# B&R Automation Studio project Soiled_PLC (part 6)

#### 12_sp2Cyclic.ab
```automation-basic
PROGRAM _CYCLIC
	(* cyclic program *)

;---------------------------------------
;Sequence 12 - SP2 Single point 2 D[912]
;---------------------------------------

;Inputs

I_BagAtBuffer			= X[9].X08
I_PaddleInPosition		= X[9].X10
I_BagInIncline			= X[9].X09
;I_BagOutAtTop           = X[7].X13

InclineEnable 		= ((D[17] > 0) AND NOT Std.HaltSys)

O_OpenBufferStop		= FALSE
O_RunMotor 				= FALSE

I_BagAtOutgoingBuffer	= FALSE
O_OutgoingBufferOpen	= FALSE

Alarm[17].Name 			= 0
Alarm[17].Bag			= 10005
Alarm[17].Beacon		= TRUE
Alarm[17].Extra			= 0
Alarm[17].Time			= 3000

;Setup Sequence
STEP = D[917]
;Setup Pulse contact
PLS = (STEP <> LASTSTEP)
LASTSTEP = STEP

;Sequence
;Step 0 - Disabled
IF (STEP = 0) THEN
	;Disabled
ENDIF

;Run Incline until paddle in position
IF (STEP = 1) THEN
	O_RunMotor = NOT I_PaddleInPosition
	IF I_PaddleInPosition THEN
		D[917] = 2
	ENDIF
	IF NOT Std.EStop THEN
		Alarm[17].Name = almSwitchFault
	ENDIF
ENDIF

;Wait for at buffer
TON_10ms(I_BagAtBuffer,300,BagAtBuffer,BagAtBufferET)
IF (STEP = 2) THEN
	IF (BagAtBuffer  AND NOT Std.HaltSys AND (D[17]>0)) THEN
		D[917] = 3
	ENDIF
	;IF (Bag[266].Cat > 0) AND NOT I_BagAtBuffer THEN
		;Alarm[12].Name 	= almBagNotAtProx
		;Alarm[12].Bag	= 266
	;ELSE IF (Bag[266].Cat = 0) AND I_BagAtBuffer THEN
		;Alarm[12].Name 	= almBagNotShownOnScreen
		;Alarm[12].Bag	= 266
	;ENDIF
ENDIF

;Open Buffer stop
IF (STEP = 3) THEN
	O_OpenBufferStop 	= TRUE
	;Enable.SIC[1]		= NOT I_BagInIncline
	IF I_BagInIncline THEN
		D[917] = 4
	ENDIF
	Alarm[17].Name = almBagNotArrived
ENDIF

;Let bag settle at base of incline
TON_10ms((STEP = 4),300,BagSettled,BagSettledET)
IF (STEP = 4) THEN
	;O_OpenBufferStop 	= TRUE
	;IF PLS THEN
	;	Bag[265] = Bag[266]
	;	Bag[266] = Bag[0]
	;ENDIF
	IF BagSettled THEN
		D[917] = 5
	ENDIF
ENDIF

;Move Bag up incline
TON_10ms((STEP = 5),700,BagNearTop,BagNearTopET)
TON_10ms(((STEP = 5) AND NOT I_BagInIncline),1000,CloseBufferStop,CloseBufferStopET)
IF (STEP = 5) THEN
	;O_OpenBufferStop 	= NOT CloseBufferStop
	O_RunMotor 			= NOT BagNearTop
	IF BagNearTop THEN
		D[917] = 6
	ENDIF
	Alarm[17].Name = almSwitchFault
ENDIF

;Check for space at destination
;Run motor for 0.5 seconds
TON_10ms((STEP = 6),50,RunOn,RunOnET)
IF (STEP = 6) THEN
	O_RunMotor 		= NOT RunOn

	IF Line[27].Clear THEN
		C[27] = 0
		D[917] = 7
	ENDIF
ENDIF

;Run incline until bag released / arrive at buffer
IF (STEP = 7) THEN
	O_RunMotor 			= TRUE
	;IF PLS THEN
	;	C[13] = 0
	;ENDIF
	IF Line[27].Trip THEN
		D[917] = 1
	ENDIF
	Alarm[17].Name = almBagNotReleased
ENDIF

;Alarms
TimerAlarm.IN 	= NOT PLS AND (Alarm[17].Name > 0)
TimerAlarm.PT 	= Alarm[17].Time
TimerAlarm FUB TON_10ms()
Alarm[17].On 	= TimerAlarm.Q
Alarm[17].ET 	= TimerAlarm.ET

;Outputs
Y[9].Y08 = O_OpenBufferStop
Y[13].Y14 = O_RunMotor
END_PROGRAM
```

### Program Logical/Sequences/10ms/18_sp6 (IEC) - * SP2 Empty bags from SDC1/2

#### 12_sp2.var
```iecst
VAR RETAIN
	STEP : UINT;
	PLS : BOOL;
	LASTSTEP : UINT;
END_VAR
VAR
	TimerAlarm : TON_10ms;
	I_BagAtBuffer : BOOL;
	O_OpenBuffer : BOOL;
	SDC2BufferFullET : TIME;
	SDC2BufferFull : BOOL;
	SettledBufferET : TIME;
	SettledBuffer : BOOL;
	O_OpenSP2BufferStop : BOOL;
	O_SelectPoint : BOOL;
	SP2BufferFull : BOOL;
	SP2BufferFullET : UDINT;
	ParingLoopEnabled : BOOL;
	BagInLoopHasDest : BOOL;
	BagAtBuffer : BOOL;
	SettledBufferSVC1 : BOOL;
	SettledBufferSVC1ET : UDINT;
	SettledBufferSVC2 : BOOL;
	SettledBufferSVC2ET : UDINT;
	O_SelectPointSVC1 : BOOL;
	O_SelectPointSVC2 : BOOL;
	I_BagatBuffer : BOOL;
	I_BagAtSVC1BufferStop : BOOL;
	I_BagAtSVC2BufferStop : BOOL;
	O_SVC1BufferStop : BOOL;
	O_SVC2BufferStop : BOOL;
	O_SelectSVC1 : BOOL;
	O_SelectSVC2 : BOOL;
	Alernate : USINT;
	BagAtBufferET : UDINT;
END_VAR
```

#### 12_sp2Cyclic.ab
```automation-basic
PROGRAM _CYCLIC
	(* cyclic program *)

;---------------------------------------
;Sequence 8 - SP8 Single point 2 D[912]
;---------------------------------------

;Inputs

I_BagatBuffer			= X[8].X11
I_BagAtSVC1BufferStop   = X[3].X06
I_BagAtSVC2BufferStop   = X[3].X14

O_SVC1BufferStop        = Y[3].Y06
O_SVC2BufferStop        = Y[3].Y14

O_OpenBuffer			= FALSE ;YB12
O_SelectSVC1            = FALSE ;YB11
O_SelectSVC2            = FALSE ;YB10

Alarm[18].Name 			= 0
Alarm[18].Bag			= 10006
Alarm[18].Beacon		= TRUE
Alarm[18].Extra			= 0
Alarm[18].Time			= 3000

;Setup Sequence
STEP = D[918]
;Setup Pulse contact
PLS = (STEP <> LASTSTEP)
LASTSTEP = STEP

;Sequence
;Step 0 - Disabled
IF (STEP = 0) THEN
	;Disabled
ENDIF

;Step 1 - decide where to take bag from
TON_10ms(I_BagatBuffer,300,BagAtBuffer,BagAtBufferET)
IF (STEP = 1) THEN

	IF BagAtBuffer THEN
	IF (Alernate > 2) THEN
		Alernate = 0
	ENDIF
	Alernate = Alernate + 1
			IF ((Alernate = 1)AND Line[28].Clear AND NOT I_BagAtSVC1BufferStop AND NOT O_SVC1BufferStop) THEN
				C[28]  = 0
				D[918] = 2
			ELSE IF ((Alernate = 2)AND Line[29].Clear AND NOT I_BagAtSVC2BufferStop AND NOT O_SVC2BufferStop) THEN
				C[29]  = 0
				D[918] = 3
			ENDIF
	ENDIF
ENDIF

;Step 2 - Bag from svc1
IF (STEP = 2) THEN
	O_OpenBuffer = TRUE
	O_SelectSVC1 = TRUE
	IF Line[28].Trip THEN
		D[918] = 1
	ENDIF
	Alarm[18].Name = almBagNotArrived
ENDIF

;Step 2 - Bag from svc1
IF (STEP = 3) THEN
	O_OpenBuffer = TRUE
	O_SelectSVC2 = TRUE
	IF Line[29].Trip THEN
		D[918] = 1
	ENDIF
	Alarm[8].Name = almBagNotArrived
ENDIF

;Alarms
TimerAlarm.IN 	= NOT PLS AND (Alarm[18].Name > 0)
TimerAlarm.PT 	= Alarm[18].Time
TimerAlarm FUB TON_10ms()
Alarm[18].On 	= TimerAlarm.Q
Alarm[18].ET 	= TimerAlarm.ET

;Outputs
Y[8].Y11 = O_OpenBuffer
Y[8].Y12 = O_SelectSVC1
Y[8].Y13 = O_SelectSVC2
END_PROGRAM
```

### Program Logical/Sequences/10ms/19_sp7 (IEC) - * SP2 Empty bags from SDC1/2

#### 12_sp2.var
```iecst
VAR RETAIN
	STEP : UINT;
	PLS : BOOL;
	LASTSTEP : UINT;
END_VAR
VAR
	TimerAlarm : TON_10ms;
	I_BagAtBuffer : BOOL;
	O_OpenBuffer : BOOL;
	SDC2BufferFullET : TIME;
	SDC2BufferFull : BOOL;
	SettledBufferET : TIME;
	SettledBuffer : ARRAY[0..2] OF BOOL;
	O_OpenSP2BufferStop : BOOL;
	O_SelectPoint : BOOL;
	SP2BufferFull : BOOL;
	SP2BufferFullET : UDINT;
	ParingLoopEnabled : BOOL;
	BagInLoopHasDest : BOOL;
	O_OpenSDC1BufferStop : BOOL;
	BagSettledAtBuffer : BOOL;
	BagSettledAtBufferET : UDINT;
	Alternator : USINT;
	BagAtBuffer : ARRAY[0..2] OF BOOL;
	SettledBufferDC1 : BOOL;
	SettledBufferDC1ET : UDINT;
	SettledBufferSD2 : BOOL;
	SettledBufferDC2ET : UDINT;
	SettledBufferDC2 : BOOL;
	I_BagAtSVC1BufferStop : BOOL;
	I_BagAtSVC2BufferStop : BOOL;
	Reset : BOOL;
	ResetET : UDINT;
	BagAtSVC1BufferStop : BOOL;
	BagAtSVC1BufferStopET : UDINT;
	BagAtSVC2BufferStop : BOOL;
	BagAtSVC2BufferStopET : UDINT;
	Alernate : USINT;
	O_SelectSVC1 : BOOL;
	O_SelectSVC2 : BOOL;
END_VAR
```

#### 12_sp2Cyclic.ab
```automation-basic
PROGRAM _CYCLIC
	(* cyclic program *)

;---------------------------------------
;Sequence 12 - SP2 Single point 2 D[912]
;---------------------------------------

;Inputs

I_BagAtSVC1BufferStop   = X[9].X05
I_BagAtSVC2BufferStop   = X[9].X06

O_OpenSDC1BufferStop	= FALSE
O_SelectPoint       	           = FALSE
O_SelectSVC1                      = FALSE
O_SelectSVC2                      = FALSE

Alarm[19].Name 			= 0
Alarm[19].Bag			= 10012
Alarm[19].Beacon	    = TRUE
Alarm[19].Extra			= 0
Alarm[19].Time			= 3000

;Setup Sequence
STEP = D[919]
;Setup Pulse contact

PLS = (STEP <> LASTSTEP)
LASTSTEP = STEP

;Sequence
;Step 0 - Disabled
IF (STEP = 0) THEN
	;Disabled
ENDIF

;Step 1 - decide where to take bag from
TON_10ms((STEP = 1),300,Reset,ResetET)
IF (STEP = 1) THEN

	IF Reset THEN
		D[919] = 2
	ENDIF
ENDIF

;Wait for Bag at buffer and destination clear
TON_10ms(I_BagAtSVC1BufferStop,300,BagAtSVC1BufferStop,BagAtSVC1BufferStopET)
TON_10ms(I_BagAtSVC2BufferStop,300,BagAtSVC2BufferStop,BagAtSVC2BufferStopET)
IF (STEP = 2) THEN
	IF (Request.SP[7] = TRUE) THEN
	IF (Alernate > 2) THEN
		Alernate = 0
	ENDIF
	Alernate = Alernate + 1
			IF ((Alernate = 1)AND BagAtSVC1BufferStop) THEN
				D[919] = 3
			ELSE IF ((Alernate = 2)AND BagAtSVC2BufferStop) THEN
				D[919] = 4
			ENDIF
	ENDIF
ENDIF

;Enable release
IF ((STEP = 3) OR (STEP = 4)) THEN
		Enable.SP[7] = TRUE
	ELSE
		Enable.SP[7] = FALSE
ENDIF

;Open buffer stop and point
IF (STEP = 3) THEN
	O_SelectSVC1 = TRUE
	IF (NOT Request.SP[7]) THEN
		D[919] = 1
	ENDIF
	Alarm[19].Name = almBagNotArrived
ENDIF

;select svc 2 point and stop
IF (STEP = 4) THEN
	O_SelectSVC2 = TRUE
	IF (NOT Request.SP[7]) THEN
		D[919] = 1
	ENDIF
	Alarm[9].Name = almBagNotArrived
ENDIF
;Alarms
TimerAlarm.IN 	= NOT PLS AND (Alarm[19].Name > 0)
TimerAlarm.PT 	= Alarm[19].Time
TimerAlarm FUB TON_10ms()
Alarm[19].On 	= TimerAlarm.Q
Alarm[19].ET 	= TimerAlarm.ET

;Outputs
Y[9].Y05 = O_SelectSVC1
Y[9].Y06 = O_SelectSVC2
END_PROGRAM
```

### Program Logical/Sequences/10ms/20_sp1 (IEC) - * SP2 Empty bags from SDC1/2

#### 12_sp2.var
```iecst
VAR RETAIN
	STEP : UINT;
	PLS : BOOL;
	LASTSTEP : UINT;
END_VAR
VAR
	TimerAlarm : TON_10ms;
	I_BagAtBuffer : BOOL;
	O_OpenBuffer : BOOL;
	SDC2BufferFullET : TIME;
	SDC2BufferFull : BOOL;
	SettledBufferET : TIME;
	SettledBuffer : BOOL;
	O_OpenSP2BufferStop : BOOL;
	O_SelectPoint : BOOL;
	SP2BufferFull : BOOL;
	SP2BufferFullET : UDINT;
	ParingLoopEnabled : BOOL;
	BagInLoopHasDest : BOOL;
	BagAtBuffer : BOOL;
	SettledBufferSVC1 : BOOL;
	SettledBufferSVC1ET : UDINT;
	SettledBufferSVC2 : BOOL;
	SettledBufferSVC2ET : UDINT;
	O_SelectPointSVC1 : BOOL;
	O_SelectPointSVC2 : BOOL;
	Reset : BOOL;
	ResetET : UDINT;
	I_BagatBuffer : BOOL;
	BagAtBufferET : UDINT;
	Alernate : USINT;
	I_BagAtSVC1BufferStop : BOOL;
	O_SVC1BufferStop : BOOL;
	I_BagAtSVC2BufferStop : BOOL;
	O_SVC2BufferStop : BOOL;
	O_SelectSVC1 : BOOL;
	O_SelectSVC2 : BOOL;
END_VAR
```

#### 12_sp2Cyclic.ab
```automation-basic
PROGRAM _CYCLIC
	(* cyclic program *)

;---------------------------------------
;Sequence 8 - SP8 Single point 2 D[912]
;---------------------------------------

;Inputs

O_SelectSVC1              = FALSE ;YB11
O_SelectSVC2              = FALSE ;YB10

Alarm[20].Name 			= 0
Alarm[20].Bag			= 221
Alarm[20].Beacon		= TRUE
Alarm[20].Extra			= 0
Alarm[20].Time			= 5000

;Setup Sequence
STEP = D[920]
;Setup Pulse contact
PLS = (STEP <> LASTSTEP)
LASTSTEP = STEP

;Sequence
;Step 0 - Disabled
IF (STEP = 0) THEN
	;Disabled
ENDIF

;clear data
TON_10ms((STEP = 1),100,Reset,ResetET)
IF (STEP = 1) THEN
	IF (Reset = TRUE)and (Bag[221].Cat = 0) THEN
		D[920] = 2
	ENDIF
ENDIF

;Wait SLU1 request and destination clear
TON_10ms(I_BagatBuffer,300,BagAtBuffer,BagAtBufferET)
IF (STEP = 2) THEN
	IF (Request.LU[1] = TRUE) THEN
	IF (Alernate > 2) THEN
		Alernate = 0
	ENDIF
	Alernate = Alernate + 1
			IF ((Alernate = 1)AND Line[30].Clear AND (Bag[223].Cat =0) AND NOT I_BagAtSVC1BufferStop AND NOT O_SVC1BufferStop) THEN
				C[30]  = 0
				D[45]  = 1
				D[920] = 3
			ELSE IF ((Alernate = 2)AND Line[18].Clear AND (Bag[222].Cat =0) AND NOT I_BagAtSVC2BufferStop AND NOT O_SVC2BufferStop) THEN
				C[18]  = 0
				D[45]  = 2
				D[920] = 4
			ENDIF
	ENDIF
ENDIF

;enable slu1 to release
IF ((STEP = 3) OR (STEP = 4)) THEN
	Enable.LU[1] = TRUE
	ELSE
	Enable.LU[1] = FALSE
ENDIF

;Open buffer to release a bag to svc 1
IF (STEP = 3) THEN

	O_SelectSVC1 = TRUE

	IF Line[30].Trip THEN
		IF (Bag[221].Cat > 0) AND (Bag[223].Cat= 0) THEN
			Bag[223] = Bag[221]
			Bag[221] = Bag[0]
		ENDIF
			D[920] = 1
	ENDIF
	Alarm[20].Name 	= almBagNotArrived
ENDIF

;select svc 2 point
IF (STEP = 4) THEN
O_SelectSVC2 = TRUE

	IF Line[18].Trip THEN
		IF (Bag[221].Cat > 0) AND (Bag[222].Cat= 0) THEN
			Bag[222] = Bag[221]
			Bag[221] = Bag[0]
		ENDIF
		D[920] = 1
	ENDIF
	Alarm[20].Name 	= almBagNotArrived
ENDIF

;Outputs

Y[9].Y07 = O_SelectSVC1
Y[9].Y12 = O_SelectSVC2

;Alarms
TimerAlarm.IN 	= NOT PLS AND (Alarm[20].Name > 0)
TimerAlarm.PT 	= Alarm[20].Time
TimerAlarm FUB TON_10ms()
Alarm[20].On 	= TimerAlarm.Q
Alarm[20].ET 	= TimerAlarm.ET

;Outputs
;Y[6].Y07 = O_SelectPointSVC1
;Y[6].Y08 = O_SelectPointSVC2
END_PROGRAM
```

### Program Logical/Sequences/10ms/10_sb1_ref (IEC, version 2.00.0) - *FROM OLD PROGRAM__ REF ONLY

#### 2_belt1Cyclic.ab
```automation-basic
PROGRAM _CYCLIC
 	(* cyclic program *)

;Sequence 2 - Transfer Belt 1 from Stations 1-12

;-----------------------------------------
;Revision 1.00 18/01/2006 D.J. First Issue
;-----------------------------------------

;Inputs and Outputs
;------------------

;Bank 						= 1

I_PhotoBottomSDC1LoadDropped = X[3].X09
I_PhotoMiddleBelt  			 = X[3].X12
I_PhotocellAtEnd             = X[5].X16
I_OpenBag                    = X[3].X05
I_LoadDropped                = X[3].X06

Enable.SDC1Drop          	= FALSE

O_RunBelt 					= FALSE
O_BagReady                  = FALSE

Alarm[10].Name 				= 0
Alarm[10].Bag				= 160
Alarm[10].Beacon			= TRUE
Alarm[10].Extra				= 0
Alarm[10].Time				= 5000

STEP = D[910]
;Setup Pulse contact
PLS = (STEP <> LASTSTEP)
LASTSTEP = STEP

;Step 0 - Disabled
IF STEP = 0 THEN
	;Disabled
ENDIF

;Step 1 - Run belt till clear
TON_10ms(((STEP = 1) AND NOT I_PhotoBottomSDC1LoadDropped AND NOT I_PhotoMiddleBelt AND NOT I_PhotocellAtEnd),500,BeltClear,BeltClearET)
IF STEP = 1 THEN
	O_RunBelt = TRUE
	IF BeltClear THEN

			D[910] = 2 ;No Bag on belt

	ENDIF
	Alarm[10].Time = 10000
	Alarm[10].Name = almPhotocellBlocked
ENDIF

;Step 2 - Wait for SDC 1 to request to drop
IF STEP = 2 THEN

		;------Write Report------
		IF Std.StationReports  THEN

			IF (ReportLoading[n].Cat = 0) THEN

				;Check if anything has been added and current weight is not less than the previous
				WeightValue = Stn[n].Weight - INT(StnPrev[n].Wgt)
				WeightValid = (WeightValue > 0)

				IF WeightValid THEN

					;Ensure valid values as we report on either a weight or count change
					IF (WeightValue < 0) THEN
						WeightValue = 0
					ENDIF

					ReportLoading[n].Cat = UINT(Bag[StnBag].Cat)	;Category
					ReportLoading[n].Cus = Bag[StnBag].Cus			;Customer
					ReportLoading[n].Wgt = UINT(WeightValue)		;Weight
					ReportLoading[n].Cnt = 0						;Count
					ReportLoading[n].Stn = n         				;Station
					ReportLoading[n].Mcn = 0						;Machine

				ENDIF

			ENDIF

		ENDIF
		IF Request.SDC1Drop THEN
			D[910] = 3
		ENDIF

		Alarm[10].Name = almNoAlarm

ENDIF

;Step 3
;Open Bag and Release to Belt Conveyor
IF STEP = 3 THEN
	Enable.SDC1Drop = TRUE
	O_RunBelt       = TRUE
	IF I_PhotoBottomSDC1LoadDropped THEN
		Bag[160] = Bag[151]

	ENDIF
	IF (Bag[160].Cat > 0) AND NOT Request.SDC1Drop AND I_PhotoBottomSDC1LoadDropped THEN
		D[910] = 4
	ENDIF
	Alarm[10].Name = almLoadNotDropped
ENDIF

;Step 4 - Run Belt Till middle
IF STEP = 4 THEN
	O_RunBelt = TRUE
	IF I_PhotoMiddleBelt THEN
		D[910] = 5
	ENDIF
	;Alarm[2].Name = almNoAlarm
ENDIF

;Step 5 - Check second bag is pair
IF STEP = 5 THEN
	;O_RunBelt = TRUE
	IF Request.SDC1Drop AND (Bag[151].Cat = Bag[160].Cat) THEN
		Bag[160].Wgt = Bag[160].Wgt + Bag[151].Wgt
		D[910] = 6
	ELSE IF Request.SDC1Drop AND (Bag[151].Cat <> Bag[160].Cat) THEN
		D[910] = 7
	ENDIF
	;Alarm[2].Name = almPhotocellNotMade
ENDIF

;Step 6 - oPEN sdc1 bag
IF STEP = 6 THEN
	Enable.SDC1Drop = TRUE
	O_RunBelt       = TRUE
	IF I_PhotoBottomSDC1LoadDropped AND NOT Request.SDC1Drop THEN
		D[910] = 7
	ENDIF
ENDIF

CodeStep  = ((STEP >= 7) AND (STEP <= 8))

IF CodeStep THEN
;round up weight to give to wash machine
;	Remainder = SINT(Bag[280].Wgt MOD 10)
;	IF (Remainder > 4) THEN
;		WgtRound = (Bag[280].Wgt + 10)
;	ELSE
;		WgtRound = Bag[280].Wgt
;	ENDIF

BCD_BIN_CAT.RegisterIN 	= Bag[160].Cat
BCD_BIN_CAT.Enable		= CodeStep
BCD_BIN_CAT.BIN			= FALSE
BCD_BIN_CAT FUB BCD_BIN_OUTPUT()

Y[9].Y05 = BCD_BIN_CAT.Output1
Y[9].Y06 = BCD_BIN_CAT.Output2
Y[9].Y07 = BCD_BIN_CAT.Output4
Y[9].Y08 = BCD_BIN_CAT.Output8
Y[9].Y09 = BCD_BIN_CAT.Output10
Y[9].Y10 = BCD_BIN_CAT.Output20
Y[9].Y11 = BCD_BIN_CAT.Output40
Y[9].Y12 = BCD_BIN_CAT.Output80

;BCD_BIN_CUS.RegisterIN 	= Bag[160].Cus
;BCD_BIN_CUS.Enable		= CodeStep
;BCD_BIN_CUS.BIN			= false
;BCD_BIN_CUS FUB BCD_BIN_OUTPUT()
;
;Y[23].Y09 = BCD_BIN_CUS.Output1
;Y[23].Y10 = BCD_BIN_CUS.Output2
;Y[23].Y11 = BCD_BIN_CUS.Output4
;Y[23].Y12 = BCD_BIN_CUS.Output8
;Y[23].Y13 = BCD_BIN_CUS.Output10
;Y[23].Y14 = BCD_BIN_CUS.Output20
;Y[23].Y15 = BCD_BIN_CUS.Output40
;Y[23].Y16 = BCD_BIN_CUS.Output80
;Y[24].Y01 = BCD_BIN_CUS.Output100
;Y[24].Y02 = BCD_BIN_CUS.Output200
;Y[24].Y03 = BCD_BIN_CUS.Output400
;Y[24].Y04 = BCD_BIN_CUS.Output800

BCD_BIN_WGT.RegisterIN 	= (Bag[160].Wgt )
BCD_BIN_WGT.Enable		= CodeStep
BCD_BIN_WGT.BIN			= false
BCD_BIN_WGT FUB BCD_BIN_OUTPUT()

Y[9].Y13 = BCD_BIN_WGT.Output1
Y[9].Y14 = BCD_BIN_WGT.Output2
Y[9].Y15 = BCD_BIN_WGT.Output4
Y[9].Y16 = BCD_BIN_WGT.Output8
Y[10].Y01 = BCD_BIN_WGT.Output10
Y[10].Y02 = BCD_BIN_WGT.Output20
Y[10].Y03 = BCD_BIN_WGT.Output40
Y[10].Y04 = BCD_BIN_WGT.Output80
Y[10].Y05 = BCD_BIN_WGT.Output100
Y[10].Y06 = BCD_BIN_WGT.Output200
Y[10].Y07 = BCD_BIN_WGT.Output400
Y[10].Y08 = BCD_BIN_WGT.Output800
ENDIF

;Step 7 - Run Belt until linen detected for 1 second and Station has emptied
TON_10ms(((STEP = 7) AND I_PhotoTop),100,LinenDetected,LinenDetectedET)
IF STEP = 7 THEN
	O_RunBelt = TRUE

	IF I_PhotocellAtEnd  THEN
		D[910] = 8
	ENDIF
	;Alarm[2].Name = almPhotocellNotMade
ENDIF

;Step 8 - Run Belt until photocells clear for 5 seconds

IF STEP = 8 THEN
	O_BagReady = TRUE
	IF I_OpenBag THEN
		D[910] = 9
	ENDIF
;	IF NOT Std.EStopLoading THEN
;		IF I_PhotoBottom OR I_PhotoTop THEN
;			Alarm[10].Name = almPhotocellBlocked
;		ELSE IF (D[901] <> 0) THEN
;			Alarm[10].Name = almStationNotClosed
;		ELSE IF NOT MinBeltRun THEN
;			Alarm[10].Name = almClearingBeltPleaseWait
;		ENDIF
;	ENDIF
ENDIF

;Step 9 - Check Stations Are Closed
IF STEP = 9 THEN
	O_RunBelt = TRUE
	IF I_LoadDropped THEN

		Bag[160] = Bag[0]
		D[910] = 1
	ENDIF
	Alarm[10].Name = almLoadNotDropped
ENDIF

;Alarms
TimerAlarm.IN = NOT PLS AND (Alarm[10].Name > 0)
TimerAlarm.PT = Alarm[10].Time
TimerAlarm FUB TON_10ms()
Alarm[10 ].On = TimerAlarm.Q
Alarm[2].ET = TimerAlarm.ET

;Outputs

Y[7].Y09 = O_BagReady

Y[7].Y06 = O_RunBelt
END_PROGRAM
```

#### 2_belt1.var
```iecst
VAR RETAIN
	MinBeltRunCV : UINT;
	MinBeltRun : BOOL;
	BeltClearET : TIME;
	BeltClear : BOOL;
	LinenDetectedET : TIME;
	LinenDetected : BOOL;
	n : UINT;
	STEP : UINT;
	Step6ET : TIME;
	LASTSTEP : UINT;
	PLS : BOOL;
	O_RunBelt : BOOL;
	RunBelt : BOOL;
END_VAR
VAR
	TimerAlarm : TON_10ms;
	I_PhotoBottom : BOOL;
	I_PhotoTop : BOOL;
	Bank : UINT;
	WeightValid : BOOL;
	WeightValue : INT;
	BeltRunTime : UINT;
	BeltAddTime : UINT;
	StnBag : UINT;
	I_PhotoBottomSDC1LoadDropped : BOOL;
	I_PhotoMiddleBelt : BOOL;
	I_PhotocellAtEnd : BOOL;
	CodeStep : BOOL;
	BCD_BIN_CAT : BCD_BIN_OUTPUT;
	BCD_BIN_WGT : BCD_BIN_OUTPUT;
	I_OpenBag : BOOL;
	I_LoadDropped : BOOL;
	O_BagReady : BOOL;
END_VAR
```

### Program Logical/Sequences/10ms/30_fvc1 (IEC) - * SVC1 Up from SLU1 & Loading

#### 8_svc1.var
```iecst
VAR RETAIN
	I_CarrAtTop : BOOL;
	I_CarrAtBottom : BOOL;
	STEP : UINT;
	PLS : BOOL;
	LASTSTEP : UINT;
	O_MoveCarrUp : BOOL;
	O_OpenCarrStop : BOOL;
	O_MoveCarrDown : BOOL;
	I_BagOnCarr : BOOL;
END_VAR
VAR
	O_OpenBuffer : BOOL;
	BagSettledOnCarr : BOOL;
	BagSettledOnCarrET : TIME;
	I_BagReleased : BOOL;
	TimerAlarm : TON_10ms;
	I_CarrAtMiddle : BOOL;
	I_CarrAtWeighing : BOOL;
	I_NoEmptyBag : BOOL;
	I_CollectEmpty : BOOL;
	I_UseAsLoading : BOOL;
	I_UpPushButton : BOOL;
	I_DownPushButton : BOOL;
	Dst : UINT;
	PButton : BOOL;
	SVCRaw : DINT;
	n : UINT;
	ValidCus : BOOL;
	ValidWgt : BOOL;
	O_AlarmLamp : BOOL;
	ValidCat : BOOL;
	Choice : ARRAY[0..4] OF UINT;
	PButtonET : TIME;
	Status : UINT;
	PastMiddleET : TIME;
	PastMiddle : BOOL;
	ValidDst : BOOL;
	I_CarrAtEmtyBagIn : BOOL;
	I_CarrAtEmptyBagOut : BOOL;
	I_FullBagReleased : BOOL;
	I_EmptyBagReleased : BOOL;
	I_FullBagAtBuffer : BOOL;
	I_WeighBeamOverRide : BOOL;
	O_MoveCarrDownToBottom : BOOL;
	O_MoveCarrDownToEmptyIn : BOOL;
	O_MoveCarrDownToEmptyBagOut : BOOL;
	OpenBufferStop : BOOL;
	NoEmptyBag : BOOL;
	BagSettledAtStop : BOOL;
	weighbeambag : INT;
	OverWeight : BOOL;
	OVERLOAD : UINT;
	LowWeight : UINT;
	UnderWeight : BOOL;
	BagSettledAtStopET : UDINT;
	WeightOK : BOOL;
	WeightOKET : UDINT;
	I_BagAtBuffer : BOOL;
	I_CarrAtEBagIn : BOOL;
	I_CarrAtSafety : BOOL;
	I_LoadingSequence : BOOL;
	I_UnLoadingSequence : BOOL;
	O_OpenBufferStop : BOOL;
	O_MoveCarrDown2 : BOOL;
	O_FVCSetpoint : BOOL;
	Beacon : BOOL;
	SignalTime : BOOL;
	SignalTimeET : UDINT;
	EBagReady : BOOL;
	EBagReadyET : UDINT;
	BagSetteled : BOOL;
	BagSetteledET : UDINT;
END_VAR
```

#### 8_svc1Cyclic.ab
```automation-basic
PROGRAM _CYCLIC
	(* cyclic program *)

;--------------------------------------------
;Sequence 8 - SVC1 Vertical conveyor 1 D[908]
;--------------------------------------------

;Inputs
I_CarrAtTop				= X[11].X02
I_CarrAtBottom			= X[11].X01
I_CarrAtEBagIn			= X[11].X03
I_CarrAtSafety			= X[11].X04
I_BagOnCarr				= X[11].X09
I_BagAtBuffer			= X[11].X11
I_UpPushButton			= X[11].X05
I_DownPushButton		= X[11].X06
I_LoadingSequence		= X[11].X07
I_UnLoadingSequence		= X[11].X08

O_OpenBufferStop		= FALSE ; YB02

;-----SAFETY CARD---------------
O_MoveCarrUp			= FALSE ; YD15
O_MoveCarrDown			= FALSE ; YD16
O_MoveCarrDown2			= FALSE ; YE01
O_OpenCarrStop			= FALSE ; YE02
O_FVCSetpoint           = FALSE

Alarm[30].Name 			= 0
Alarm[30].Bag			= 315
Alarm[30].Beacon		= TRUE
Alarm[30].Extra			= 0
Alarm[30].Time			= 3000

;Setup Sequence
STEP = D[930]
;Setup Pulse contact
PLS = (STEP <> LASTSTEP)
LASTSTEP = STEP

;Sequence
IF (STEP = 0) THEN
	;Disabled
ENDIF

;show bag on screen
IF (STEP >= 1) AND (STEP <= 4) THEN
	Bag[315] = Bag[321]
;	E[1571] = E[1601]
ENDIF

;Move Carriage down to loading position
IF (STEP = 1) THEN
O_MoveCarrDown = ((I_CarrAtBottom = FALSE) AND (I_DownPushButton = TRUE))
	IF (I_CarrAtBottom = TRUE) THEN
		D[930] = 2
	ENDIF
	IF NOT Std.EStop THEN
		Alarm[16].Name = almCarriageMoveFault
	ENDIF
ENDIF

;Bag loading
;Move Carriage up to safety level
IF (STEP = 2) THEN
	O_MoveCarrDown = ((I_CarrAtBottom = FALSE) AND (I_DownPushButton = TRUE) AND (I_UpPushButton = FALSE))
	O_MoveCarrUp = ((I_CarrAtSafety = FALSE) AND (I_DownPushButton = FALSE) AND (I_UpPushButton = TRUE))
	IF (I_CarrAtSafety = TRUE) THEN
		D[930] = 3
	ENDIF
ENDIF

;Check neither push button is pressed
IF (STEP = 3) THEN
	IF ((I_UpPushButton = FALSE) AND (I_DownPushButton = FALSE)) THEN
		D[930] = 4
	ENDIF
ENDIF

;Check Destination Clear and up push button pressed
TON_10ms(((STEP = 4) AND (I_UpPushButton = TRUE)),50,PButton,PButtonET)
IF (STEP = 4) THEN
	 Bag[315].Cat = Bag[310].Cat
	Bag[315].Cus = Bag[310].Cus
	Bag[315].Prg = usint(Bag[310].Cat)

    IF ((I_BagOnCarr = TRUE) AND (PButton = TRUE) AND (Bag[315].Cat > 0)) THEN
		;Update Bag ID if cleared or zero
		IF ((BidStn > 0) AND (Bag[315].Bid = 0) AND (Bag[315].Cat > 0)) THEN
			Bag[315].Bid = UINT(BidStn)
			BidStn			= 0
		ENDIF
		D[930] = 5
	ENDIF
ENDIF

;Reset sequence if Down push button pressed
IF ((STEP = 4) AND (I_DownPushButton = TRUE)) THEN
	D[930] = 1
ENDIF

;Select Unloading sequence
IF ((STEP = 4) AND (I_BagOnCarr = FALSE) AND (I_UnLoadingSequence = TRUE)) THEN
	IF (PButton = TRUE) THEN
		D[930] = 13
	ENDIF
ENDIF

;Move Carriage up to top position
IF (STEP = 5) THEN
	O_MoveCarrUp = (I_CarrAtTop = FALSE)
	IF (I_CarrAtTop = TRUE) THEN
		D[930] = 6
	ENDIF
ENDIF

;Wait for Release bag signal
TON_10ms((STEP = 6),200,SignalTime,SignalTimeET)
IF (STEP = 6) THEN
    IF ((Line[41].Clear = TRUE) AND (Bag[308].Cat = 0)) THEN
		D[930] = 7
		C[41]  = 0
	ENDIF
ENDIF

;Releasing onto storage
IF (STEP = 7) THEN
	O_OpenCarrStop = (I_CarrAtTop = TRUE)
	D[58]     = 1

	;Bag at destination
	IF (Line[41].Trip = TRUE) THEN
		IF (Bag[315].Cat >0) AND (Bag[308].Cat =0) THEN
			Bag[308] = Bag[315]
			Bag[315] = Bag[0]
		ENDIF
		D[930] = 8
	ENDIF

	Alarm[30].Name = almBagNotReleased
ENDIF

;Move Carriage down to empty position
IF (STEP = 8) THEN
	O_MoveCarrDown2 = ((I_CarrAtEBagIn = FALSE) AND (I_CarrAtBottom = FALSE))
	IF (I_CarrAtEBagIn = TRUE) THEN
		D[930] = 9
	ENDIF
	Alarm[30].Name = almCarriageMoveFault
ENDIF

;Wait for empty bag to settle
;Or Loading program selected
TON_10ms(((I_BagAtBuffer = TRUE) AND (I_BagOnCarr = FALSE) AND (STEP = 9)),100,EBagReady,EBagReadyET)
IF (STEP = 9) THEN
	IF (EBagReady = TRUE) AND (I_BagAtBuffer = TRUE) THEN
		D[930] = 10
	ENDIF
	IF (I_LoadingSequence = TRUE) THEN
		D[930] = 12
	ENDIF
ENDIF

;Bag at buffer stop
IF (STEP = 10) THEN
	O_OpenBufferStop = (I_CarrAtEBagIn = TRUE)
	D[58]     = 2
	IF (I_BagOnCarr = TRUE) THEN
		D[930] = 11
	ENDIF
	Alarm[30].Name = almBagNotReleased
	ELSE
	O_OpenBufferStop = FALSE
ENDIF

;bag settles on carriage
TON_10ms((I_BagOnCarr = TRUE),300,BagSetteled,BagSetteledET)
IF (STEP = 11) THEN
	IF (BagSetteled = TRUE) THEN
		D[930] = 12
	ENDIF
ENDIF

;Move Carriage down to safety position
IF (STEP = 12) THEN
	O_MoveCarrDown = ((I_CarrAtSafety = FALSE) AND (I_CarrAtBottom = FALSE))
	IF (I_CarrAtSafety = TRUE) THEN
		D[930] = 1
	ENDIF
ENDIF

;-------------------------------
;-----UNLOADING PROGRAM---------
;-------------------------------
IF (STEP = 13) THEN
	O_MoveCarrUp = (I_CarrAtTop = FALSE)
	IF (I_CarrAtTop = TRUE) THEN
		D[930] = 8
	ENDIF
ENDIF

;Alarms
TimerAlarm.IN 	= NOT PLS AND (Alarm[30].Name > 0)
TimerAlarm.PT 	= Alarm[30].Time
TimerAlarm FUB TON_10ms()
Alarm[30].On 	= TimerAlarm.Q
Alarm[30].ET 	= TimerAlarm.ET

;PLC Outputs
;-----------

Y[11].Y02 = (O_OpenBufferStop AND (I_CarrAtEBagIn = TRUE ))

;-------SAFETY CARD-------------
Y[13].Y15 = ((O_MoveCarrUp = TRUE) AND (I_CarrAtTop = FALSE))
Y[13].Y16 = ((O_MoveCarrDown = TRUE) AND (I_CarrAtBottom = FALSE))
Y[14].Y01 = ((O_MoveCarrDown2 = TRUE) AND (I_CarrAtBottom = FALSE) AND (I_CarrAtEBagIn = FALSE))
Y[14].Y02 = ((O_OpenCarrStop = TRUE) AND (I_CarrAtTop = TRUE))

;Don't allow forcing of carriage movement and carriage stop
YForceDisable[13].Y15 = TRUE
YForceDisable[13].Y16 = TRUE
YForceDisable[14].Y01 = TRUE
YForceDisable[14].Y02 = TRUE

END_PROGRAM
```

### Program Logical/Sequences/10ms/ssr (IEC, version 1.00.1) - speed reducer

#### ssr.st - Implementation code
```iecst
(********************************************************************
 * COPYRIGHT --
 ********************************************************************
 * Program: ssr
 * File: ssr.st
 * Author: treamsbottom
 * Created: July 16, 2015
 ********************************************************************
 * Implementation of program ssr
 ********************************************************************)
//V1.00.1 FIRST VERSION
PROGRAM _INIT

END_PROGRAM

PROGRAM _CYCLIC

;myHaltSys				:= Std.HaltSysZone[0];

//Inputs
i_bagApproach[1]		:= X[4].X16;
i_bagApproach[2]		:= X[4].X07;
FOR n := 1 TO LOCAL_MAX_SPEED_REDUCERS DO

	ctu_tripCount[n](CU	:= i_bagApproach[n],PV := 2,RESET := ton_10ms_openBrush[n].Q);
	ton_10ms_openBrush[n](IN :=  o_closeBrush[n],PT	:= 600);

	IF (ctu_tripCount[n].CV >= 1) THEN
		o_closeBrush[n] := TRUE;
	END_IF;

	IF ton_10ms_openBrush[n].Q THEN
		o_closeBrush[n] := FALSE;
	END_IF;
END_FOR;

//Outputs
Y[5].Y15		:= o_closeBrush[1];
Y[5].Y14          := o_closeBrush[2];

END_PROGRAM
```

#### ssr.var - Local variables
```iecst
(********************************************************************
 * COPYRIGHT --
 ********************************************************************
 * Program: ssr
 * File: ssr.var
 * Author: treamsbottom
 * Created: July 16, 2015
 ********************************************************************
 * Local variables of program ssr
 ********************************************************************)
VAR
	myHaltSys : BOOL;
	i_bagApproach : ARRAY[0..LOCAL_MAX_SPEED_REDUCERS] OF BOOL;
	n : UINT;
	ctu_tripCount : ARRAY[0..LOCAL_MAX_SPEED_REDUCERS] OF CTU;
	ton_10ms_openBrush : ARRAY[0..LOCAL_MAX_SPEED_REDUCERS] OF TON_10ms;
	o_closeBrush : ARRAY[0..LOCAL_MAX_SPEED_REDUCERS] OF BOOL;
END_VAR
VAR CONSTANT
	LOCAL_MAX_SPEED_REDUCERS : UINT := 2;
END_VAR
VAR
	kev : BOOL;
END_VAR
```

### Program Logical/Sequences/10ms/31_fdc1 (IEC) - * SDC1 Machine 1 BIN/BCD

#### 6_sdc1Cyclic.ab
```automation-basic
PROGRAM _CYCLIC
	(* cyclic program *)

;Sequence 6 - Discharger 1 D[906]

;-----------------------------------------
;Revision 1.00 19/12/2005 D.J. First Issue
;-----------------------------------------

DischargerEnable 		= ((D[16] > 0) AND NOT Std.HaltSys)

I_ReadyToLoad           = X[12].X01 OR TestLoad
I_OpenBag				= X[12].X02
I_LoadDropped			= X[12].X03
I_BagAtDischarger		= X[11].X13 OR Testxb13
I_BagOutDischarger      = X[11].X15

O_BagReady				= FALSE
O_OpenBuffer 			= FALSE
O_Steadys				= FALSE
O_OpenBag				= FALSE
O_Closer				= FALSE
O_OpenStop				= FALSE

Request.FDC[1] 			= FALSE
Request.FDCEmpty[1]     = FALSE

EndOfLoading            = FALSE
;Alarm
Alarm[31].Name 			= almNoAlarm ;Clear sequence alarm name
Alarm[31].Bag 			= 317
Alarm[31].Beacon			= TRUE
Alarm[31].Extra			= 0
Alarm[31].Time			= 3000

;Setup Sequence
STEP = D[931]
;Setup Pulse contact
PLS = (STEP <> LASTSTEP)
LASTSTEP = STEP

;Step 0 - Disabled
IF (STEP = 0) THEN
	;Disabled
ENDIF

;Check Status - Discharger clear
TON_10ms((NOT I_BagAtDischarger),200,DischargerClear,DischargerClearET)
IF (STEP = 1) THEN
	IF ((DischargerClear)  AND (D[28] > 0) AND ((Bag[317].Cat = 0) OR (D[970] > 0))) THEN
		D[931] = 2
	ENDIF
ENDIF

;Wait for bag in discharger
IF (STEP = 2) THEN
Request.FDC[1] = I_ReadyToLoad

	IF I_BagAtDischarger THEN

		IF (Bag[317].Cat = 0) THEN ;move bag into discharger if first bag
			Bag[317] = Bag[316]
			Bag[316] = Bag[0]
			D[931] = 3
		ENDIF
	ENDIF
ENDIF

;Let bag settle in discharger
;Settled At Discharger (Sad)
TON_10ms(((STEP = 3) AND I_BagAtDischarger),1000,SettledAtDischarger,SettledAtDischargerET)
IF (STEP = 3) THEN
	IF SettledAtDischarger THEN
		D[931] = 4
	ENDIF
	Alarm[31].Time = 2000
	Alarm[31].Name = almBagNotSettled
ENDIF

;Allow steadys to move down
TON_10ms((STEP = 4),400,SteadysDown,SteadysDownET)
IF (STEP = 4) THEN
	IF SteadysDown THEN
		D[931] = 5
	ENDIF
	IF (Bag[317].Cat = Std.MaxCats) THEN
		D[931] = 7
	ENDIF
ENDIF

;Steady cylinders on from steps 4 - 9
O_Steadys = ((STEP >= 4) AND (STEP <= 9))

;Bag opener on from step 5 - 8
O_OpenBag = ((STEP >= 6) AND (STEP <= 8))

CodeStep  = ((STEP >= 4) AND (STEP <= 5))

;Wash Codes
;Wash Codes
IF CodeStep THEN
;Wash Codes
BCD_BIN_CAT.RegisterIN 	= Bag[317].Cat
BCD_BIN_CAT.Enable		= CodeStep
BCD_BIN_CAT.BIN			= TRUE
BCD_BIN_CAT FUB BCD_BIN_OUTPUT()

Y[12].Y01 = BCD_BIN_CAT.Output1
Y[12].Y02 = BCD_BIN_CAT.Output2
Y[12].Y03 = BCD_BIN_CAT.Output4
Y[12].Y04 = BCD_BIN_CAT.Output8
Y[12].Y05 = BCD_BIN_CAT.Output10
;Y[10].Y14 = BCD_BIN_CAT.Output20
;Y[10].Y15 = BCD_BIN_CAT.Output40
;Y[10].Y16 = BCD_BIN_CAT.Output80

;BCD_BIN_CUS.RegisterIN 	= Bag[152].Cus
;BCD_BIN_CUS.Enable		= CodeStep
;BCD_BIN_CUS.BIN			= FALSE
;BCD_BIN_CUS FUB BCD_BIN_OUTPUT()
;
;Y[11].Y01 = BCD_BIN_CUS.Output1
;Y[11].Y02 = BCD_BIN_CUS.Output2
;Y[11].Y03 = BCD_BIN_CUS.Output4
;Y[11].Y04 = BCD_BIN_CUS.Output8
;Y[11].Y05 = BCD_BIN_CUS.Output10
;Y[11].Y06 = BCD_BIN_CUS.Output20
;Y[11].Y07 = BCD_BIN_CUS.Output40
;Y[11].Y08 = BCD_BIN_CUS.Output80
;Y[11].Y09 = BCD_BIN_CUS.Output100
;Y[11].Y10 = BCD_BIN_CUS.Output200
;Y[11].Y11 = BCD_BIN_CUS.Output400
;Y[11].Y12 = BCD_BIN_CUS.Output800

;BCD_BIN_WGT.RegisterIN 	= (Bag[152].Wgt / 10)
;BCD_BIN_WGT.Enable		= CodeStep
;BCD_BIN_WGT.BIN			= FALSE
;BCD_BIN_WGT FUB BCD_BIN_OUTPUT()
;
;Y[26].Y05 = BCD_BIN_WGT.Output1
;Y[26].Y06 = BCD_BIN_WGT.Output2
;Y[26].Y07 = BCD_BIN_WGT.Output4
;Y[26].Y08 = BCD_BIN_WGT.Output8
;Y[26].Y09 = BCD_BIN_WGT.Output10
;Y[26].Y10 = BCD_BIN_WGT.Output20
;Y[26].Y11 = BCD_BIN_WGT.Output40
;Y[26].Y12 = BCD_BIN_WGT.Output80
ELSE
Y[12].Y01 =  FALSE
Y[12].Y02 =  FALSE
Y[12].Y03 =  FALSE
Y[12].Y04 =  FALSE
Y[12].Y05=  FALSE
ENDIF

;Bag Ready to Washing Machine
IF (STEP = 5) THEN
	O_BagReady = (Bag[317].Cat > 0)
	IF I_OpenBag THEN
		D[931] = 6
	ENDIF
	IF (Bag[317].Cat = 0) THEN
		Alarm[31].Time = 1
		Alarm[31].Name = almBagNotShownOnScreen
	ENDIF
	ELSE
	O_BagReady = FALSE
ENDIF

;Set LoadDropped to False
IF (STEP <> 6) THEN
	LoadDropped = FALSE
ENDIF

;Open Bag Until LoadDropped recieved and has been open for 6 seconds
TON_10ms((STEP = 6),600,MinOpen,MinOpenET) ;ET means Elapsed Time
IF (STEP = 6) THEN

	IF I_LoadDropped OR TestDischarger THEN
	;IF I_BagEmpty THEN
		LoadDropped = TRUE
	ENDIF

	IF (LoadDropped AND MinOpen) THEN
		;Write Report
		;------------
		IF (ReportUnloading[3].Cat = 0) THEN
			ReportUnloading[3].Cat = UINT(Bag[317].Cat)	;Category
			ReportUnloading[3].Cus = Bag[317].Cus		;Customer
			ReportUnloading[3].Wgt = 500		;Weight
			ReportUnloading[3].Cnt = 0					;Count
			ReportUnloading[3].Stn = 0					;Station
			ReportUnloading[3].Mcn = 3					;Machine
		ENDIF
	ENDIF
	IF (LoadDropped AND MinOpen) THEN
		D[931] = 7
	ENDIF
	Alarm[31].Name = almLoadNotDropped
ENDIF

;Change display to empty bag
IF (STEP = 7) THEN
	IF ((D[970] = 0 AND NOT I_LoadDropped AND I_BagEmpty) OR TestDrop) THEN
		Bag[317].Prg 	= Std.MaxProg
		Bag[317].Cat 	= Std.MaxCats
		D[931] 			= 8
	ENDIF
	IF  NOT I_LoadDropped AND NOT I_OpenBag then
		D[931] 			= 8
	ENDIF
	Alarm[31].Name = almGeneralSequence
ENDIF

;Close bag
TON_10ms((STEP = 8),100,CloserDown,CloserDownET)
IF (STEP = 8) THEN
	O_Closer = TRUE
	IF CloserDown THEN
		D[931] = 9
	ENDIF
ENDIF

;Allow closer to go back up
TON_10ms((STEP = 9),100,CloserUp,CloserUpET)
IF (STEP = 9) THEN
	IF CloserUp THEN
		D[931] = 10
	ENDIF
ENDIF

;Allow steadys to go up
TON_10ms((STEP = 10),400,SteadyUp,SteadyUpET)
IF (STEP = 10) THEN
	EndOfLoading = (D[970] = 0)
	IF (SteadyUp AND NOT Enable.FDCEmpty[1])THEN
		D[931] = 11
	ENDIF
ENDIF

;Check for space on empty bag buffer
IF (STEP = 11) THEN
	Request.FDCEmpty[1] = TRUE
	IF (Enable.FDCEmpty[1] AND NOT I_BagOutDischarger) THEN
		D[931] = 12
	ENDIF
ENDIF

;Open buffer stop - unitl bag out
IF (STEP = 12) THEN
	O_OpenStop = TRUE
	Bag[317] = Bag[0]
	IF (PLS AND (D[970] = 0)) THEN
			Bag[317] = Bag[0]
	ENDIF
	IF I_BagOutDischarger THEN
		D[931] = 1
	ENDIF

	Alarm[31].Name = almBagNotReleased
ENDIF

;Alarms
TimerAlarm.IN 	= NOT PLS AND (Alarm[31].Name > 0)
TimerAlarm.PT 	= Alarm[31].Time
TimerAlarm FUB TON_10ms()
Alarm[31].On 	= TimerAlarm.Q
Alarm[31].ET 	= TimerAlarm.ET

;Outputs
Y[12].Y12            = O_BagReady
Y[11].Y03 			= O_Steadys
Y[11].Y04 			= O_OpenBag
Y[11].Y05 			= O_Closer
Y[11].Y13 			= O_OpenStop
Y[12].Y13            = EndOfLoading
END_PROGRAM
```

### Program Logical/Sequences/10ms/32_fdc2 (IEC) - * SDC1 Machine 1 BIN/BCD

#### 6_sdc1.var
```iecst
VAR RETAIN
	STEP : UINT;
	PLS : BOOL;
	LASTSTEP : UINT;
	SteadyUp : BOOL;
	CloserUpET : TIME;
	SteadysDown : BOOL;
	SteadysDownET : TIME;
	LoadDropped : BOOL;
	SteadyUpET : TIME;
	CloserDownET : TIME;
	SettledAtDischargerET : TIME;
	MinOpenET : TIME;
	SettledAtDischarger : BOOL;
	CloserDown : BOOL;
	MinOpen : BOOL;
	CloserUp : BOOL;
	SettledAtBuffer : BOOL;
	SettledAtBufferET : TIME;
	I_BagAtBuffer : BOOL;
	O_OpenStop : BOOL;
	O_OpenBag : BOOL;
	O_Steadys : BOOL;
	O_OpenBuffer : BOOL;
	O_Closer : BOOL;
	I_BagAtDischarger : BOOL;
	I_OpenBag : BOOL;
	I_LoadDropped : BOOL;
	TestDrop : BOOL;
END_VAR
VAR
	DischargerEnable : BOOL;
	TestDischarger : BOOL;
	I_BagEmpty : BOOL;
	O_BagReady : BOOL;
	I_BagReleased : BOOL;
	O_EmptyBagBufferOpen : BOOL;
	I_BagAtEmptyBuffer : BOOL;
	TimerAlarm : TON_10ms;
	CodeStep : BOOL;
	BCD_BIN_CAT : BCD_BIN_OUTPUT;
	BCD_BIN_CUS : BCD_BIN_OUTPUT;
	BCD_BIN_WGT : BCD_BIN_OUTPUT;
	Remainder : UINT;
	WgtRound : UINT;
	Weight : UINT;
	I_ReadyToLoad : BOOL;
	TestLoad : BOOL;
	Testxb13 : BOOL;
	I_BagOutDischarger : BOOL;
	EndOfLoading : BOOL;
	DischargerClear : BOOL;
	DischargerClearET : UDINT;
END_VAR
```

#### 6_sdc1Cyclic.ab
```automation-basic
PROGRAM _CYCLIC
	(* cyclic program *)

;Sequence 6 - Discharger 1 D[906]

;-----------------------------------------
;Revision 1.00 19/12/2005 D.J. First Issue
;-----------------------------------------

DischargerEnable 		= ((D[16] > 0) AND NOT Std.HaltSys)

I_ReadyToLoad           = X[12].X07
I_OpenBag				= X[12].X08
I_LoadDropped			= X[12].X09

I_BagAtDischarger		= X[11].X14
I_BagEmpty                  = TRUE
O_BagReady				= FALSE
O_OpenBuffer 			= FALSE
O_Steadys				= FALSE
O_OpenBag				= FALSE
O_Closer				= FALSE
O_OpenStop				= FALSE

Request.FDC[2] 			= FALSE
Request.FDCEmpty[2]     = FALSE

EndOfLoading            = FALSE
;Alarm
Alarm[32].Name 			= almNoAlarm ;Clear sequence alarm name
Alarm[32].Bag 			= 318
Alarm[32].Beacon			= TRUE
Alarm[32].Extra			= 0
Alarm[32].Time			= 3000

;Setup Sequence
STEP = D[932]
;Setup Pulse contact
PLS = (STEP <> LASTSTEP)
LASTSTEP = STEP

;Step 0 - Disabled
IF (STEP = 0) THEN
	;Disabled
ENDIF

;Check Status - Discharger clear
TON_10ms((NOT I_BagAtDischarger),200,DischargerClear,DischargerClearET)
IF (STEP = 1) THEN
	IF ((DischargerClear)  AND (D[28] > 0) AND ((Bag[318].Cat = 0) OR (D[971] > 0))) THEN
		D[932] = 2
	ENDIF
ENDIF

;Wait for bag in discharger
IF (STEP = 2) THEN
Request.FDC[2] = I_ReadyToLoad

	IF I_BagAtDischarger THEN
			D[932] = 3
		IF (Bag[318].Cat = 0) THEN ;move bag into discharger if first bag
			Bag[318] = Bag[316]
			Bag[316] = Bag[0]
			D[932] = 3
		ENDIF
	ENDIF
ENDIF

;Let bag settle in discharger
;Settled At Discharger (Sad)
TON_10ms(((STEP = 3) AND I_BagAtDischarger),1000,SettledAtDischarger,SettledAtDischargerET)
IF (STEP = 3) THEN
	IF SettledAtDischarger THEN
		D[932] = 4
	ENDIF
	Alarm[32].Time = 2000
	Alarm[32].Name = almBagNotSettled
ENDIF

;Allow steadys to move down
TON_10ms((STEP = 4),400,SteadysDown,SteadysDownET)
IF (STEP = 4) THEN
	IF SteadysDown THEN
		D[932] = 5
	ENDIF
	IF (Bag[318].Cat = Std.MaxCats) THEN
		D[932] = 7
	ENDIF
ENDIF

;Steady cylinders on from steps 4 - 9
O_Steadys = ((STEP >= 4) AND (STEP <= 9))

;Bag opener on from step 5 - 8
O_OpenBag = ((STEP >= 6) AND (STEP <= 8))

CodeStep  = ((STEP >= 4) AND (STEP <= 5))

;Wash Codes
;Wash Codes
IF CodeStep THEN
;Wash Codes
BCD_BIN_CAT.RegisterIN 	= Bag[318].Cat
BCD_BIN_CAT.Enable		= CodeStep
BCD_BIN_CAT.BIN			= TRUE
BCD_BIN_CAT FUB BCD_BIN_OUTPUT()

Y[12].Y06 = BCD_BIN_CAT.Output1
Y[12].Y07 = BCD_BIN_CAT.Output2
Y[12].Y08 = BCD_BIN_CAT.Output4
Y[12].Y09 = BCD_BIN_CAT.Output8
Y[12].Y10 = BCD_BIN_CAT.Output10
;Y[10].Y14 = BCD_BIN_CAT.Output20
;Y[10].Y15 = BCD_BIN_CAT.Output40
;Y[10].Y16 = BCD_BIN_CAT.Output80

;BCD_BIN_CUS.RegisterIN 	= Bag[152].Cus
;BCD_BIN_CUS.Enable		= CodeStep
;BCD_BIN_CUS.BIN			= FALSE
;BCD_BIN_CUS FUB BCD_BIN_OUTPUT()
;
;Y[11].Y01 = BCD_BIN_CUS.Output1
;Y[11].Y02 = BCD_BIN_CUS.Output2
;Y[11].Y03 = BCD_BIN_CUS.Output4
;Y[11].Y04 = BCD_BIN_CUS.Output8
;Y[11].Y05 = BCD_BIN_CUS.Output10
;Y[11].Y06 = BCD_BIN_CUS.Output20
;Y[11].Y07 = BCD_BIN_CUS.Output40
;Y[11].Y08 = BCD_BIN_CUS.Output80
;Y[11].Y09 = BCD_BIN_CUS.Output100
;Y[11].Y10 = BCD_BIN_CUS.Output200
;Y[11].Y11 = BCD_BIN_CUS.Output400
;Y[11].Y12 = BCD_BIN_CUS.Output800

;BCD_BIN_WGT.RegisterIN 	= (Bag[152].Wgt / 10)
;BCD_BIN_WGT.Enable		= CodeStep
;BCD_BIN_WGT.BIN			= FALSE
;BCD_BIN_WGT FUB BCD_BIN_OUTPUT()
;
;Y[26].Y05 = BCD_BIN_WGT.Output1
;Y[26].Y06 = BCD_BIN_WGT.Output2
;Y[26].Y07 = BCD_BIN_WGT.Output4
;Y[26].Y08 = BCD_BIN_WGT.Output8
;Y[26].Y09 = BCD_BIN_WGT.Output10
;Y[26].Y10 = BCD_BIN_WGT.Output20
;Y[26].Y11 = BCD_BIN_WGT.Output40
;Y[26].Y12 = BCD_BIN_WGT.Output80
ELSE
Y[12].Y06 =  FALSE
Y[12].Y07 =  FALSE
Y[12].Y08 =  FALSE
Y[12].Y09 =  FALSE
Y[12].Y10 =  FALSE
ENDIF

;Bag Ready to Washing Machine
IF (STEP = 5) THEN
	O_BagReady = (Bag[318].Cat > 0)
	IF I_OpenBag THEN
		D[932] = 6
	ENDIF
	IF (Bag[318].Cat = 0) THEN
		Alarm[32].Time = 10
		Alarm[32].Name = almBagNotShownOnScreen
	ENDIF
	ELSE
	O_BagReady = FALSE
ENDIF

;Set LoadDropped to False
IF (STEP <> 6) THEN
	LoadDropped = FALSE
ENDIF

;Open Bag Until LoadDropped recieved and has been open for 6 seconds
TON_10ms((STEP = 6),600,MinOpen,MinOpenET) ;ET means Elapsed Time
IF (STEP = 6) THEN

	IF I_LoadDropped OR TestDischarger THEN
	;IF I_BagEmpty THEN
		LoadDropped = TRUE
	ENDIF

	IF (LoadDropped AND MinOpen) THEN
		;Write Report
		;------------
		IF (ReportUnloading[4].Cat = 0) THEN
			ReportUnloading[4].Cat = UINT(Bag[318].Cat)	;Category
			ReportUnloading[4].Cus = Bag[318].Cus		;Customer
			ReportUnloading[4].Wgt = 500		;Weight
			ReportUnloading[4].Cnt = 0					;Count
			ReportUnloading[4].Stn = 0					;Station
			ReportUnloading[4].Mcn = 4					;Machine
		ENDIF
	ENDIF
	IF (LoadDropped AND MinOpen) THEN
		D[932] = 7
	ENDIF
	Alarm[32].Name = almLoadNotDropped
ENDIF

;Change display to empty bag
IF (STEP = 7) THEN
	IF ((NOT Enable.SDC1Drop AND NOT I_LoadDropped AND I_BagEmpty) OR TestDrop) THEN
		Bag[318].Prg 	= Std.MaxProg
		Bag[318].Cat 	= Std.MaxCats
		D[932] 			= 8
	ENDIF
	IF NOT I_OpenBag AND NOT I_LoadDropped then
		D[932] 			= 8
	ENDIF
	Alarm[31].Name = almGeneralSequence
ENDIF

;Close bag
TON_10ms((STEP = 8),100,CloserDown,CloserDownET)
IF (STEP = 8) THEN
	O_Closer = TRUE
	IF CloserDown THEN
		D[932] = 9
	ENDIF
ENDIF

;Allow closer to go back up
TON_10ms((STEP = 9),100,CloserUp,CloserUpET)
IF (STEP = 9) THEN
	IF CloserUp THEN
		D[932] = 10
	ENDIF
ENDIF

;Allow steadys to go up
TON_10ms((STEP = 10),400,SteadyUp,SteadyUpET)
IF (STEP = 10) THEN
	EndOfLoading = (D[971] = 0)
	IF (SteadyUp AND NOT Enable.FDCEmpty[1])THEN
		D[932] = 11
	ENDIF
ENDIF

;Check for space on empty bag buffer
IF (STEP = 11) THEN
	Request.FDCEmpty[2] = TRUE
	IF Enable.FDCEmpty[2] THEN
		D[932] = 12
	ENDIF
ENDIF

;Open buffer stop - unitl bag out
IF (STEP = 12) THEN
	O_OpenStop = TRUE
	Bag[318] = Bag[0]
	IF (PLS AND (D[971] = 0)) THEN

		Bag[318] = Bag[0]
	ENDIF
	IF NOT Enable.FDCEmpty[2] THEN
		D[932] = 1
	ENDIF

	Alarm[32].Name = almBagNotReleased
ENDIF

;Alarms
TimerAlarm.IN 	= NOT PLS AND (Alarm[32].Name > 0)
TimerAlarm.PT 	= Alarm[32].Time
TimerAlarm FUB TON_10ms()
Alarm[32].On 	= TimerAlarm.Q
Alarm[32].ET 	= TimerAlarm.ET

;Outputs
Y[15].Y06            = O_BagReady
Y[11].Y07 			= O_Steadys
Y[11].Y08 			= O_OpenBag
Y[11].Y09 			= O_Closer
Y[11].Y14 			= O_OpenStop
Y[15].Y07            = EndOfLoading
END_PROGRAM
```

### Program Logical/Sequences/10ms/33_fp1 (IEC, version 1.00.0) - * SP2 Empty bags from SDC1/2

#### 12_sp2Cyclic.ab
```automation-basic
PROGRAM _CYCLIC
	(* cyclic program *)

;---------------------------------------
;Sequence 12 - SP2 Single point 2 D[912]
;---------------------------------------

;Inputs

D[970] = 0
D[971] = 0

LOOP CurrentBag = Line[30].FirstBag  TO Line[30].LastBag DO
;LOOP CurrentBag = 301  TO 301 DO
		EXITIF Line[30].FirstBag = 0
		FirstBagDestination = Bag[301].Dst
		CurrentDis = (Bag[CurrentBag].Dst)
		EXITIF (FirstBagDestination <> Bag[CurrentBag].Dst)
		IF (((Bag[CurrentBag].Dst) = FirstBagDestination) AND (FirstBagDestination = 23))THEN
			D[970] = (D[970] + 1)
			testkk = TRUE
		ENDIF
		IF (((Bag[CurrentBag].Dst)= FirstBagDestination) AND (FirstBagDestination = 24))THEN
			D[971] = (D[971] + 1)
		ENDIF

ENDLOOP

Uld[3].SDCReady 	= ((D[28] > 0)AND (Request.FDC[1] = TRUE) AND (D[970] = 0) AND (Bag[316].Cat= 0))
Uld[4].SDCReady 	= ((D[29] > 0)AND (Request.FDC[2] = TRUE) AND (D[971] = 0) AND (Bag[316].Cat = 0))

I_BagAtStop 		= X[11].X12

O_OpenBufferStop    = FALSE

Alarm[33].Name 			= 0
Alarm[33].Bag			= 316
Alarm[33].Beacon		= TRUE
Alarm[33].Extra			= 0
Alarm[33].Time			= 2000

;Setup Sequence
STEP = D[933]
;Setup Pulse contact
PLS = (STEP <> LASTSTEP)
LASTSTEP = STEP

;Sequence
;Step 0 - Disabled
IF (STEP = 0) THEN
	;Disabled
ENDIF

IF I_BagAtStop  AND (Bag[301].Cat=0) THEN
	Alarm[33].Name 			= almSwitchFault
	Alarm[33].Time			= 300
ELSE IF NOT I_BagAtStop  AND (Bag[301].Cat>0) THEN
	Alarm[33].Name 			= almBagNotSettled
	Alarm[33].Time			= 10000
ENDIF

;;Step 1 - Reset Points
TON_10ms((STEP = 1),300,ResetPoints,ResetPointsET)
IF (STEP = 1) THEN
		Destination = 0
	IF ResetPoints THEN
		D[933] = 2
	ENDIF
ENDIF

;Bag at buffer stop with dest
TON_10ms((I_BagAtStop),300,BagAtBuffer,BagAtBufferET)
IF (STEP = 2) THEN
	IF BagAtBuffer THEN
		IF ((Request.FDC[1] = TRUE)AND (Bag[301].Cat > 0) AND (Bag[301].Dst= 23) AND (D[970] > 0))  THEN
			Destination = 1
			D[933] = 3

		ELSE IF ((Request.FDC[2] = TRUE) AND (Bag[301].Cat > 0) AND (Bag[301].Dst= 24) AND (D[971] > 0)) THEN
			Destination = 2
			D[933] = 3
		ENDIF
	ENDIF
ENDIF

;Select discharger
IF (STEP = 3) THEN
	O_OpenBufferStop = TRUE
	IF ((Bag[301].Cat >0) AND (Bag[316].Cat = 0) AND PLS) THEN
		Bag[316] = Bag[301]
		Bag[301] = Bag[0]
	ENDIF
	IF (D[931] > 2) AND (Destination = 1)THEN ;Bag at FDC 1
		D[933] = 1
	ELSE IF (D[932] > 2) AND (Destination = 2) THEN
		D[933] = 1
	ENDIF
	Alarm[33].Name 			= almBagNotReleased

ENDIF

;Alarms
TimerAlarm.IN 	= NOT PLS AND (Alarm[33].Name > 0)
TimerAlarm.PT 	= Alarm[33].Time
TimerAlarm FUB TON_10ms()
Alarm[33].On 	= TimerAlarm.Q
Alarm[33].ET 	= TimerAlarm.ET

;Outputs
Y[11].Y12 = O_OpenBufferStop

Y[11].Y10 = (Destination = 1);FP1
Y[11].Y11 = (Destination = 2);FP1

END_PROGRAM
```

#### 12_sp2.var
```iecst
VAR RETAIN
	STEP : UINT;
	PLS : BOOL;
	LASTSTEP : UINT;
END_VAR
VAR
	TimerAlarm : TON_10ms;
	I_BagAtBuffer : BOOL;
	O_OpenBuffer : BOOL;
	SDC2BufferFullET : TIME;
	SDC2BufferFull : BOOL;
	SettledBufferET : TIME;
	SettledBuffer : BOOL;
	O_OpenSP2BufferStop : BOOL;
	O_SelectPoint : BOOL;
	SP2BufferFull : BOOL;
	SP2BufferFullET : UDINT;
	ParingLoopEnabled : BOOL;
	BagInLoopHasDest : BOOL;
	O_OpenSDC1BufferStop : BOOL;
	BagSettledAtBuffer : BOOL;
	BagSettledAtBufferET : UDINT;
	Alternator : USINT;
	I_OnLineA : BOOL;
	I_TiltA : BOOL;
	I_TiltB : BOOL;
	I_Bagout : BOOL;
	O_OpenBufferStop : BOOL;
	O_SelectLineA : BOOL;
	O_SelectLineB : BOOL;
	O_OpenStops : BOOL;
	O_TiltCylinder : BOOL;
	O_OperatePusher : BOOL;
	PointReset : BOOL;
	PointResetET : UDINT;
	BagAtTilt : BOOL;
	BagAtTiltET : UDINT;
	TiltDown : BOOL;
	TiltDownET : UDINT;
	TiltUp : BOOL;
	TiltUpET : UDINT;
	NotFull : BOOL;
	NotFullET : UDINT;
	Pushed : BOOL;
	SBSN1 : BOOL;
	SBSN1ET : UDINT;
	RequirePusherET : UDINT;
	PushedET : UDINT;
	I_BagAtBufferStop : BOOL;
	O_SP7ToSVC1 : BOOL;
	O_SP7ToSIC3 : BOOL;
	SDC1EmptyBufferFull : BOOL;
	SDC1EmptyBufferFullET : UDINT;
	Reset : BOOL;
	ResetET : UDINT;
	ResetPoint : BOOL;
	CurrentBag : UINT;
	FirstBagDestination : USINT;
	CurrentDis : USINT;
	E : BOOL;
	I_BagAtStop : BOOL;
	ResetPoints : BOOL;
	ResetPointsET : UDINT;
	BagAtBuffer : BOOL;
	BagAtBufferET : UDINT;
	Destination : USINT;
	test : BOOL;
	testkk : BOOL;
END_VAR
```

### Program Logical/Sequences/10ms/34_fp2 (IEC) - * SP2 Empty bags from SDC1/2

#### 12_sp2.var
```iecst
VAR RETAIN
	STEP : UINT;
	PLS : BOOL;
	LASTSTEP : UINT;
END_VAR
VAR
	TimerAlarm : TON_10ms;
	I_BagAtBuffer : BOOL;
	O_OpenBuffer : BOOL;
	SDC2BufferFullET : TIME;
	SDC2BufferFull : BOOL;
	SettledBufferET : TIME;
	SettledBuffer : BOOL;
	O_OpenSP2BufferStop : BOOL;
	O_SelectPoint : BOOL;
	SP2BufferFull : BOOL;
	SP2BufferFullET : UDINT;
	ParingLoopEnabled : BOOL;
	BagInLoopHasDest : BOOL;
	O_OpenSDC1BufferStop : BOOL;
	BagSettledAtBuffer : BOOL;
	BagSettledAtBufferET : UDINT;
	Alternator : USINT;
	I_OnLineA : BOOL;
	I_TiltA : BOOL;
	I_TiltB : BOOL;
	I_Bagout : BOOL;
	O_OpenBufferStop : BOOL;
	O_SelectLineA : BOOL;
	O_SelectLineB : BOOL;
	O_OpenStops : BOOL;
	O_TiltCylinder : BOOL;
	O_OperatePusher : BOOL;
	PointReset : BOOL;
	PointResetET : UDINT;
	BagAtTilt : BOOL;
	BagAtTiltET : UDINT;
	TiltDown : BOOL;
	TiltDownET : UDINT;
	TiltUp : BOOL;
	TiltUpET : UDINT;
	NotFull : BOOL;
	NotFullET : UDINT;
	Pushed : BOOL;
	SBSN1 : BOOL;
	SBSN1ET : UDINT;
	RequirePusherET : UDINT;
	PushedET : UDINT;
	I_BagAtBufferStop : BOOL;
	O_SP7ToSVC1 : BOOL;
	O_SP7ToSIC3 : BOOL;
	SDC1EmptyBufferFull : BOOL;
	SDC1EmptyBufferFullET : UDINT;
	Reset : BOOL;
	ResetET : UDINT;
	ResetPoint : BOOL;
END_VAR
```

#### 12_sp2Cyclic.ab
```automation-basic
PROGRAM _CYCLIC
	(* cyclic program *)

;---------------------------------------
;Sequence 12 - SP2 Single point 2 D[912]
;---------------------------------------

;Inputs

O_OpenBufferStop		 = FALSE ;Y714
ResetPoint				        = FALSE ;Y711

Enable.FDCEmpty[1]      = FALSE
Enable.FDCEmpty[2]      = FALSE

Alarm[34].Name 		    	= 0
Alarm[34].Bag		    	= 10011
Alarm[34].Beacon		= TRUE
Alarm[34].Extra		    	= 0
Alarm[34].Time			   = 3000

;Setup Sequence
STEP = D[934]
;Setup Pulse contact
PLS = (STEP <> LASTSTEP)
LASTSTEP = STEP

;Sequence
;Step 0 - Disabled
IF (STEP = 0) THEN
	;Disabled
ENDIF

;reset data
TON_10ms((STEP = 1),200,Reset,ResetET)
IF (STEP = 1) THEN

	ResetPoint = TRUE
	IF Reset THEN
		D[934] = 2
	ENDIF
ENDIF

;bag at discharger
IF (STEP = 2) THEN
	IF (Line[42].Clear = TRUE) THEN
		IF (Request.FDCEmpty[1] = TRUE) THEN
			C[42] = 0
			D[934] = 3
		ELSE IF (Request.FDCEmpty[2] = TRUE) THEN
			C[42] = 0
			D[934] = 4

		ENDIF
	ENDIF
ENDIF

;select FDC 1
IF (STEP = 3) THEN
		Enable.FDCEmpty[1] = TRUE

	IF (Line[42].Trip = TRUE)  THEN
		D[934] = 1

	ENDIF
ENDIF

;select FDC 2
IF (STEP = 4) THEN
	 Enable.FDCEmpty[2] = TRUE

	IF (Line[42].Trip = TRUE)  THEN
		D[934] = 1

	ENDIF
ENDIF

;Alarms
TimerAlarm.IN 	= NOT PLS AND (Alarm[34].Name > 0)
TimerAlarm.PT 	= Alarm[34].Time
TimerAlarm FUB TON_10ms()
Alarm[34].On 	= TimerAlarm.Q
Alarm[34].ET 	= TimerAlarm.ET

END_PROGRAM
```

### Program Logical/Sequences/10ms/35_fpr1 (IEC) - * SP2 Empty bags from SDC1/2

#### 12_sp2.var
```iecst
VAR RETAIN
	STEP : UINT;
	PLS : BOOL;
	LASTSTEP : UINT;
END_VAR
VAR
	TimerAlarm : TON_10ms;
	I_BagAtBuffer : BOOL;
	O_OpenBuffer : BOOL;
	SDC2BufferFullET : TIME;
	SDC2BufferFull : BOOL;
	SettledBufferET : TIME;
	SettledBuffer : BOOL;
	O_OpenSP2BufferStop : BOOL;
	O_SelectPoint : BOOL;
	SP2BufferFull : BOOL;
	SP2BufferFullET : UDINT;
	ParingLoopEnabled : BOOL;
	BagInLoopHasDest : BOOL;
	O_OpenSDC1BufferStop : BOOL;
	BagSettledAtBuffer : BOOL;
	BagSettledAtBufferET : UDINT;
	Alternator : USINT;
	I_PaddleInPosition : BOOL;
	I_BagInIncline : BOOL;
	O_OpenBufferStop : BOOL;
	O_RunMotor : BOOL;
	I_BagAtOutgoingBuffer : BOOL;
	O_OutgoingBufferOpen : BOOL;
	BagSettled : BOOL;
	BagSettledET : UDINT;
	BagNearTop : BOOL;
	BagNearTopET : UDINT;
	CloseBufferStop : BOOL;
	CloseBufferStopET : UDINT;
	RunOn : BOOL;
	RunOnET : UDINT;
	I_BagOutAtTop : BOOL;
	BagAtBuffer : BOOL;
	BagAtBufferET : UDINT;
	I_BagStackerNearFull : BOOL;
	BagStackerHasSpace : BOOL;
	BagStackerHasSpaceET : UDINT;
	SIC3BufferFull : BOOL;
	SIC3BufferFullET : UDINT;
	HaltDownStairs : BOOL;
	SPL1BufferOpen : BOOL;
	SPITransitBag : BOOL;
	BagSettle : BOOL;
	BagSettleET : UDINT;
	SettledAtBuffer : BOOL;
	SettledAtBufferET : UDINT;
END_VAR
```

#### 12_sp2Cyclic.ab
```automation-basic
PROGRAM _CYCLIC
	(* cyclic program *)

;---------------------------------------
;Sequence 12 - SP2 Single point 2 D[912]
;---------------------------------------

;Inputs

I_BagAtBuffer        = X[10].X13

O_OpenBufferStop     = FALSE

STEP = D[935]
;Setup Pulse contact
PLS = (STEP <> LASTSTEP)
LASTSTEP = STEP

;Alarm
Alarm[35].Name 			= 0
Alarm[35].Bag			= 310
Alarm[35].Beacon		= TRUE
Alarm[35].Extra			= 0
Alarm[35].Time			= 3000

TON_10ms(I_BagAtBuffer,300,SettledAtBuffer,SettledAtBufferET)
IF (STEP = 1) THEN
    IF ((SettledAtBuffer) AND (I_BagAtBuffer = TRUE) AND (Line[43].Clear = TRUE)) THEN
    D[935] = 2
  ENDIF
ENDIF

;Wait For Bag Out
IF (STEP = 2) THEN
 O_OpenBufferStop = TRUE
   IF PLS THEN
      C[43] = 0
ENDIF
   IF (C[43]>= 1) THEN
   D[935] = 1
  ENDIF

 	Alarm[35].Name = almBagNotArrived
ENDIF

;Alarms
TimerAlarm.IN 	= NOT PLS AND (Alarm[35].Name > 0)
TimerAlarm.PT 	= Alarm[35].Time
TimerAlarm FUB TON_10ms()
Alarm[35].On 	= TimerAlarm.Q
Alarm[35].ET 	= TimerAlarm.ET

Y[10].Y13 = O_OpenBufferStop

END_PROGRAM
```

### Program Logical/Sequences/10ms/36_sb_a (IEC) - * SP2 Empty bags from SDC1/2

#### 12_sp2.var
```iecst
VAR RETAIN
	STEP : UINT;
	PLS : BOOL;
	LASTSTEP : UINT;
END_VAR
VAR
	TimerAlarm : TON_10ms;
	I_BagAtBuffer : BOOL;
	O_OpenBuffer : BOOL;
	SDC2BufferFullET : TIME;
	SDC2BufferFull : BOOL;
	SettledBufferET : TIME;
	SettledBuffer : BOOL;
	O_OpenSP2BufferStop : BOOL;
	O_SelectPoint : BOOL;
	SP2BufferFull : BOOL;
	SP2BufferFullET : UDINT;
	ParingLoopEnabled : BOOL;
	BagInLoopHasDest : BOOL;
	O_OpenSDC1BufferStop : BOOL;
	BagSettledAtBuffer : BOOL;
	BagSettledAtBufferET : UDINT;
	Alternator : USINT;
	I_OnLineA : BOOL;
	I_TiltA : BOOL;
	I_TiltB : BOOL;
	I_Bagout : BOOL;
	O_OpenBufferStop : BOOL;
	O_SelectLineA : BOOL;
	O_SelectLineB : BOOL;
	O_OpenStops : BOOL;
	O_TiltCylinder : BOOL;
	O_OperatePusher : BOOL;
	PointReset : BOOL;
	PointResetET : UDINT;
	BagAtTilt : BOOL;
	BagAtTiltET : UDINT;
	TiltDown : BOOL;
	TiltDownET : UDINT;
	TiltUp : BOOL;
	TiltUpET : UDINT;
	NotFull : BOOL;
	NotFullET : UDINT;
	Pushed : BOOL;
	SBSN1 : BOOL;
	SBSN1ET : UDINT;
	RequirePusherET : UDINT;
	PushedET : UDINT;
	I_BagAtBufferStop : BOOL;
	O_SP7ToSVC1 : BOOL;
	O_SP7ToSIC3 : BOOL;
	SDC1EmptyBufferFull : BOOL;
	SDC1EmptyBufferFullET : UDINT;
	Reset : BOOL;
	ResetET : UDINT;
	ResetPoint : BOOL;
	WasherUnloading : BOOL;
	Testwash : BOOL;
	ManaulOperation : BOOL;
	InchPushButton : BOOL;
	BeltA_DetectsLargeLoad : BOOL;
	SBA_PhotocellReverse : BOOL;
	SBA_Photocell : BOOL;
	SB_3PhotocellFullBottom : BOOL;
	SB4_PhotoCell : BOOL;
	LoadOK : BOOL;
	O_BrakeA : BOOL;
	O_BrakeSB3 : BOOL;
	O_BeltReadyFDC1 : BOOL;
	O_BeltReadyFDC2 : BOOL;
	AlarmLamp : BOOL;
	O_OK_Lamp : BOOL;
	O_ReverseBeltA : BOOL;
	O_RunBeltA_Slow : BOOL;
	O_RunBeltA_Forward : BOOL;
	O_RunBeltB_Forward : BOOL;
	O_RunBeltB_Slow : BOOL;
	O_RunBeltB_Speed2 : BOOL;
	O_Runbelt3_Forward : BOOL;
	O_Runbelt3_Slow : BOOL;
	O_RunBelt3_Speed2 : BOOL;
	O_PauseUnloading : BOOL;
	AlarmET : UDINT;
	StopBelts : BOOL;
	ResetBelt : BOOL;
	ResetBeltET : UDINT;
	Alternate : INT;
	FDC1 : BOOL;
	FDC1ET : UDINT;
	Clear : BOOL;
	ClearET : UDINT;
	FDC2 : BOOL;
	FDC2ET : UDINT;
	Clear1 : BOOL;
	Clear1ET : UDINT;
	RunBelt : BOOL;
	StopBeltET : UDINT;
	RunBeltET : UDINT;
	SB_3Full : BOOL;
	SB_3FullET : UDINT;
	SB_3Clear : BOOL;
	SB_3ClearET : UDINT;
	LinenDetected : BOOL;
	LinenDetectedET : UDINT;
	I_SafetyRelayOn : BOOL;
	SB2Clear : BOOL;
	SB2ClearET : UDINT;
	SBBeltClear : BOOL;
	SBBeltClearET : UDINT;
	SlowA : BOOL;
	BeltAlarm : BOOL;
	Slow1 : BOOL;
	Slow1ET : UDINT;
	SlowB : BOOL;
	Slow3 : BOOL;
	SlowAET : UDINT;
	SlowBET : UDINT;
	Slow3ET : UDINT;
	kev : BOOL;
END_VAR
```

#### 12_sp2Cyclic.ab
```automation-basic
PROGRAM _CYCLIC
	(* cyclic program *)

;---------------------------------------
;Sequence 12 - SP2 Single point 2 D[912]
;---------------------------------------

;Inputs

WasherUnloading         = X[12].X04 OR Testwash;relay in panel signal from washers
ManaulOperation         = X[12].X16;switch on remote box
InchPushButton          = X[12].X12;momentery push button

BeltA_DetectsLargeLoad  = X[12].X14;photocell on belt SB-A
SBA_PhotocellReverse    = X[12].X10;photocell at end of SB-A in reverse

SBA_Photocell           = X[12].X15;linen detected end of SB-A
SB_3PhotocellFullBottom = X[12].X11;linen at end of conveyor when reversing

SB4_PhotoCell           = X[12].X13;

LoadOK                  = X[15].X01;push button on panel

O_BrakeA                = FALSE
O_BrakeSB3              = FALSE

O_BeltReadyFDC1         = FALSE;relay to washer
O_BeltReadyFDC2         = FALSE;relay to washer

AlarmLamp               = FALSE ;Lamp on panel
O_OK_Lamp               = FALSE ;lamp in push button

O_ReverseBeltA          = FALSE
O_RunBeltA_Slow         = FALSE
O_RunBeltA_Forward      = FALSE ;speed 2
O_RunBeltB_Forward      = FALSE ;speed 1
O_RunBeltB_Slow         = FALSE ;speed 1
O_RunBeltB_Speed2       = FALSE
O_Runbelt3_Forward      = FALSE
O_Runbelt3_Slow         = FALSE
O_RunBelt3_Speed2       = FALSE
O_PauseUnloading        = FALSE

Request.SB[2]           = FALSE

Alarm[36].Name 			= 0
Alarm[36].Bag			= 10009
Alarm[36].Beacon		= TRUE
Alarm[36].Extra			= 0
Alarm[36].Time			= 3000

;Setup Sequence
STEP = D[936]
;Setup Pulse contact
PLS = (STEP <> LASTSTEP)
LASTSTEP = STEP

;Alarm

IF ((STEP >= 3) AND (STEP <= 6)) OR ((STEP >=7) AND (STEP <= 10)) THEN
    O_BrakeA = TRUE
ELSE
    O_BrakeA = FALSE
ENDIF

IF ((STEP >= 4) AND (STEP <= 9) AND (STEP <> 5) AND NOT StopBelts)  THEN
    O_BrakeSB3 = TRUE
ELSE
    O_BrakeSB3 = FALSE
ENDIF

;Sequence
IF (STEP = 0) THEN
	;disabled
ENDIF

TON_10ms(((STEP = 1)),200,ResetBelt,ResetBeltET)
IF (STEP = 1) THEN
	IF ResetBelt THEN
		D[936] = 2
	ENDIF
ENDIF

IF STEP <> 2 THEN
	Alternate = 1
ENDIF

;Wait for unload signal and manaul or auto
TON_10ms(((STEP = 2) AND (Alternate = 1)),500,FDC1,FDC1ET)
TON_10ms(((STEP = 2)AND (Alternate = 2)),200,Clear,ClearET)
TON_10ms(((STEP = 2)AND (Alternate = 3)),500,FDC2,FDC2ET)
TON_10ms(((STEP = 2)AND (Alternate = 4)),200,Clear1,Clear1ET)
IF (STEP = 2) THEN
	IF ((Alternate > 4) OR (Alternate <= 0)) THEN
		 Alternate = 1
    ENDIF

    IF FDC1 THEN
    	Alternate = 2
    ELSE IF Clear THEN
    	Alternate = 3
    ELSE IF FDC2 THEN
    	Alternate = 4
	ELSE IF Clear1 THEN
		Alternate = 1
	ENDIF

	O_BeltReadyFDC1 = (Alternate = 1)
    O_BeltReadyFDC2 = (Alternate = 3)

	;O_BeltReadyFDC1 = Std.M9035
	;O_BeltReadyFDC2 = NOT Std.M9035

	IF ((WasherUnloading = TRUE) AND (NOT ManaulOperation)) THEN
		D[936] = 4 ;changed from 3
	ELSE IF ((WasherUnloading = TRUE) AND  (ManaulOperation = TRUE)) THEN
		D[936] = 10
	ENDIF
ENDIF

;run belt at 10 meters a minute
IF (STEP = 3) THEN
	O_RunBeltA_Forward = TRUE ;10ms
	IF (BeltA_DetectsLargeLoad = TRUE) THEN
		D[936] = 7
	ENDIF
	IF (SBA_Photocell = TRUE) THEN
		D[936] = 4
	ENDIF
ENDIF

TON_10ms((STEP = 6) AND NOT RunBelt,500,StopBelts,StopBeltET)
TON_10ms(StopBelts,500,RunBelt,RunBeltET)

TON_10ms((SB_3PhotocellFullBottom = TRUE),50,SB_3Full,SB_3FullET)
TON_10ms((SB_3PhotocellFullBottom = FALSE),50,SB_3Clear,SB_3ClearET)
TON_10ms(((STEP = 4) AND SB4_PhotoCell),600,LinenDetected,LinenDetectedET)
IF (STEP = 4) THEN
	;IF NOT StopBelts THEN
	     O_RunBeltA_Forward   = TRUE ;SB_3Clear
	     O_RunBeltA_Slow      = kev
	     O_RunBeltB_Forward   = TRUE
	     O_RunBeltB_Speed2    = TRUE
	     O_Runbelt3_Forward   = TRUE
	     O_RunBelt3_Speed2    = TRUE
	 ;ENDIF
	IF (BeltA_DetectsLargeLoad = TRUE) THEN
		D[936] = 8
	ENDIF
	IF (LinenDetected = TRUE) THEN
		D[936] = 5
	ENDIF
ENDIF

;I_SafetyRelayOn and sb2 not running
TON_10ms(((NOT Std.HaltSys AND (Y[14].Y04= TRUE) AND (NOT Y[14].Y03) )),1700,SB2Clear,SB2ClearET)
IF (STEP = 5) THEN
	Request.SB[2] = TRUE
	IF (SB2Clear = TRUE) THEN
		D[936] = 6
	ENDIF
ENDIF

;run belts at 10ms
TON_10ms(((STEP = 6) AND (NOT SB4_PhotoCell) AND (NOT Std.HaltSys = TRUE)),3000,SBBeltClear,SBBeltClearET)
IF (STEP = 6) THEN
		Request.SB[2] = TRUE
    IF ((Y[14].Y04 = TRUE) AND NOT StopBelts) THEN
		 O_RunBeltA_Forward         = TRUE
		 O_RunBeltA_Slow            = SlowA
		 O_RunBeltB_Forward         = TRUE
		 O_Runbelt3_Forward         = TRUE
	ENDIF
	IF (BeltA_DetectsLargeLoad = TRUE) THEN
		BeltAlarm   = TRUE
		D[936] = 9
	ENDIF
	IF SBBeltClear THEN
		D[936] = 1
	ENDIF
ENDIF

;Large load from step 3
IF (STEP = 7) THEN
	AlarmLamp              = TRUE
	O_OK_Lamp              = TRUE
	O_PauseUnloading       = TRUE
	IF (InchPushButton AND (SB4_PhotoCell = FALSE)) THEN
	    O_RunBeltA_Forward = TRUE

		O_RunBeltA_Slow    = Slow1

	ENDIF
	IF LoadOK THEN
		D[936] = 3
	ENDIF
ENDIF

TON_10ms((O_RunBeltA_Forward = TRUE),50,Slow1,Slow1ET)

;Large load from step 4
IF (STEP = 8) THEN
	AlarmLamp              = TRUE
	O_OK_Lamp              = TRUE
	O_PauseUnloading       = TRUE
	IF (InchPushButton AND (SB4_PhotoCell = FALSE)) THEN
	    O_RunBeltA_Forward = TRUE
	    O_RunBeltA_Slow    = SlowA
	    O_RunBeltB_Forward = TRUE
	    O_RunBeltB_Slow    = SlowB
	    O_Runbelt3_Forward = TRUE
	    O_Runbelt3_Slow    = Slow3

	ENDIF
	IF LoadOK THEN
		D[936] = 4
	ENDIF
  ENDIF

;Large load from step 6
IF (STEP = 9) THEN
	AlarmLamp              = TRUE
	O_OK_Lamp              = TRUE
	O_PauseUnloading       = TRUE
	IF (InchPushButton AND (SB4_PhotoCell = FALSE)) THEN
		O_RunBeltA_Slow    = SlowA
	    O_RunBeltA_Forward = TRUE
	    O_RunBeltB_Forward = TRUE
	    O_RunBeltB_Slow    = SlowB
	    O_Runbelt3_Forward = TRUE
	    O_Runbelt3_Slow    = Slow3

	ENDIF
	IF LoadOK THEN
		D[936] = 6
	ENDIF
ENDIF

;manual mode
IF (STEP = 10) THEN
	;AlarmLamp              = TRUE
	O_OK_Lamp              = TRUE
	;O_PauseUnloading       = TRUE
	IF (InchPushButton  AND (SBA_PhotocellReverse = FALSE)) THEN
	    O_ReverseBeltA    = TRUE
	ENDIF
	IF LoadOK THEN
		D[936] = 1
	ENDIF
ENDIF

TON_10ms((O_RunBeltA_Forward = TRUE),50,SlowA,SlowAET)
TON_10ms((O_RunBeltB_Forward = TRUE),50,SlowB,SlowBET)
TON_10ms((O_Runbelt3_Forward = TRUE),50,Slow3,Slow3ET)
;Alarms
TimerAlarm.IN 	= NOT PLS AND (Alarm[36].Name > 0)
TimerAlarm.PT 	= Alarm[36].Time
TimerAlarm FUB TON_10ms()
Alarm[36].On 	= TimerAlarm.Q
Alarm[36].ET 	= TimerAlarm.ET

;Outputs
Y[12].Y15 = AlarmLamp ;YC15
Y[15].Y01 = O_OK_Lamp ;Lamp on push button box YF01
Y[12].Y14  = O_BeltReadyFDC1;YC14
Y[12].Y16  = O_BeltReadyFDC2;YC16

Y[14].Y13= O_RunBeltA_Slow ;YE13
Y[14].Y09 = O_RunBeltA_Forward;YE09

Y[14].Y11 = O_RunBeltB_Forward;YE11

Y[14].Y05 = O_Runbelt3_Forward  ;YYE05

Y[14].Y12 = O_RunBeltB_Slow;YE12

Y[14].Y08 = O_Runbelt3_Slow ;YE08

Y[14].Y10 = O_ReverseBeltA    ;YE10

Y[15].Y02 = O_RunBeltB_Speed2 ;YF02

Y[15].Y03 = O_RunBelt3_Speed2 ;YF03

Y[15].Y04 = O_PauseUnloading  ;YF04

Y[14].Y06 = Y[14].Y05

Y[14].Y16 = O_BrakeA ;YE16
Y[14].Y14 = O_BrakeSB3  ;YE14
END_PROGRAM
```

### Program Logical/Sequences/10ms/12_PN2 (IEC) - *Ongoing Sequence

#### x_pn.ab
```automation-basic
PROGRAM _CYCLIC

;--------------------------------------
;Sequence 4 - Ongoing To Storage D[900 + mySeq]
;--------------------------------------

;--------------------------------------------------------------------------------
;Revision 1.00 06/11/2009 D.J. First Issue - Automatic Line Allocation with Areas
;--------------------------------------------------------------------------------
mySeq 			= 12
myZone 			= 0
myTransitBag	= 297
myStartStop		= 100

IF (myStartStop >= 100) THEN
	myStartStop = myStartStop + 7600
ENDIF

;Inputs
OnGoingEnable 		= ((D[25] > 0) AND NOT Std.HaltSysZone[myZone])

I_BagatBuffer[1]		= Request.VC[2]
I_BagatBuffer[2]		= FALSE
I_BagatBuffer[3]		= FALSE
I_BagatBuffer[4]		= FALSE

O_Reset 		  		= FALSE
O_OpenSelect[1]			= FALSE
O_OpenSelect[2]			= FALSE
O_OpenSelect[3]			= FALSE
O_OpenSelect[4]			= FALSE

O_OpenBuffer[1]			= FALSE
O_OpenBuffer[2]			= FALSE
O_OpenBuffer[3]			= FALSE
O_OpenBuffer[4]			= FALSE

MaxBuffers 			= 1 	;Set Max Buffers to search
MinLine				= 1 	;Set First Storage Line
MaxLine				= 5		;Set Last Storage Line
MaxDepth			= 9    ;Capacity of the longest line - used in search

Alarm[mySeq].Name 		= 0
Alarm[mySeq].Bag		= myTransitBag
Alarm[mySeq].Beacon		= TRUE
Alarm[mySeq].Extra	 	= 0
Alarm[mySeq].Time		= 6000

;Setup Sequence
;--------------
STEP = D[900 + mySeq]
;Setup Pulse contact
PLS = (STEP <> LASTSTEP)
LASTSTEP = STEP

;Step 0 - Disabled
IF (STEP = 0) THEN
	;Disabled
ENDIF

;Step 1 - Reset Ongoing Points
TON_10ms((STEP = 1),300,ResetPoints,ResetPointsET)
IF (STEP = 1) THEN
	Dest  	= 0
	Buff 	= 0
	O_Reset = TRUE
	IF (ResetPoints AND OnGoingEnable) THEN
		D[900 + mySeq] = 2
	ENDIF
ENDIF

;Bag Settles at each buffer
TON_10ms(Request.SVC3LowLevel,100,SettledBuffer[1],SettledBufferET[1])       ;sequence 10 on step 13(SVC3)
TON_10ms(Request.SVC2FullBagLowLevel,100,SettledBuffer[2],SettledBufferET[2])  ;sequence 9 on step 13(SVC2)
;TON_10ms(I_BagatBuffer[3],300,SettledBuffer[3],SettledBufferET[3])

MaxBuffers = 2
BufferBagNum[1]	= 310
BufferBagNum[2]	= 296
;BufferBagNum[3]	= myTransitBag

;Step 2 - Search for a valid Bag at one of the buffers
IF (STEP = 2) THEN

	Buff 	= 0
	Dest 	= 0

	IF OnGoingEnable THEN

		Alarm[mySeq].Name 	= almNoAlarm

		;Search only 1 buffer bag per scan/task
		Buffer = Buffer + 1
		IF Buffer > MaxBuffers THEN
			Buffer = 1
		ENDIF
		;Set Test Value for Monitoring
		IF TestBuffer > 0 THEN
			Buffer = TestBuffer
		ENDIF

		BufferBag		= BufferBagNum[Buffer]
		BufferSettled 	= SettledBuffer[Buffer]
		BufferPrg 		= Bag[BufferBag].Prg
		BufferCat		= Bag[BufferBag].Cat
		BufferCus		= Bag[BufferBag].Cus
		BufferDst 		= Bag[BufferBag].Dst

		IF (BufferSettled AND (BufferCat > 0) AND (BufferPrg > 0) AND (BufferPrg <= Std.MaxProg) AND (OnGoingEnable)) THEN

			;Manual Destination has been set?
			IF (BufferDst > 0) THEN

				n = BufferDst
				IF ((n >= MinLine) AND (n <= MaxLine) AND (Line[n].Space > 0) AND Line[n].Clear) THEN
					Dest 	= n
					Buff 	= Buffer
					D[900 + mySeq] 	= 3
				ELSE
					Alarm[mySeq].Name 	= almDestinationNotValid
					Alarm[mySeq].Bag	= BufferBag
				ENDIF

			ELSE IF Std.AutoLineAllocation THEN ;/BufferDst > 0

				;Search Each Storage Area
				AreaChoice[1] = D[3000 + BufferPrg]
				AreaChoice[2] = D[3100 + BufferPrg]
				AreaChoice[3] = D[3200 + BufferPrg]
				AreaChoice[4] = D[3300 + BufferPrg]

				LOOP Area = 1 TO 4 DO

					AreaStartLine 	= D[250 + AreaChoice[Area]]
					AreaEndLine 	= D[270 + AreaChoice[Area]]
					AreaValid		= ((AreaStartLine > 0) AND (AreaEndLine > 0) AND (AreaEndLine >= AreaStartLine))
					IF AreaValid THEN

						;Search for a line with the same program
						;---------------------------------------
						LOOP myLine = AreaStartLine TO AreaEndLine DO
							myLineValid = ((myLine >= MinLine) AND (myLine <= MaxLine))
							myLineUsed	= (D[myStartStop + myLine] > 0) ;Start / Stop On
							IF myLineValid AND myLineUsed THEN
								n 			= myLine
								SearchBag 	= (Line[n].LastBag - Line[n].Space)
								IF ((SearchBag >= Line[n].FirstBag) AND (Bag[SearchBag].Prg = BufferPrg) AND (Line[n].Space > 0) AND Line[n].Clear) THEN
									;Found line with a matching program
									Dest 	= n
								ENDIF ;/SearchBag
							ENDIF ;/myLineValid
							EXITIF (Dest <> 0)
						ENDLOOP ;/myLine loop

						;Search for an empty line
						;------------------------
						IF (Dest = 0) THEN
							LOOP myLine = AreaStartLine TO AreaEndLine DO
								myLineValid = ((myLine >= MinLine) AND (myLine <= MaxLine))
								myLineUsed	= (D[myStartStop + myLine] > 0) ;Start / Stop On
								IF myLineValid AND myLineUsed THEN
									n 			= myLine
									SearchBag 	= (Line[n].FirstBag)
									IF ((Bag[SearchBag].Prg = 0) AND (Line[n].Space > 0) AND Line[n].Clear) THEN
										;Found line with a matching program
										Dest 	= n
									ENDIF ;/SearchBag
								ENDIF ;/myLineValid
							EXITIF (Dest <> 0)
							ENDLOOP ;/myLine loop
						ENDIF ;/Dest = 0

						;Search for a line that already contains a bag with the same program starting at the back
						;----------------------------------------------------------------------------------------
						IF (Dest = 0) THEN
							LOOP myDepth = (MaxDepth - 2) DOWNTO 0 DO ;Don't search the last bag as the line would already be full!!
								LOOP myLine = AreaStartLine TO AreaEndLine DO
									myLineValid = ((myLine >= MinLine) AND (myLine <= MaxLine))
									myLineUsed	= (D[myStartStop + myLine] > 0) ;Start / Stop On
									IF myLineValid AND myLineUsed THEN
										n 			= myLine
										SearchBag 	= (Line[n].FirstBag + myDepth)
										IF ((Bag[SearchBag].Prg = BufferPrg) AND (Line[n].Space > 0) AND Line[n].Clear) THEN
											;Found line with a matching program
											FoundDepth 	= myDepth
											Dest 		= n
										ENDIF ;/SearchBag
									ENDIF ;/myLineValid
									EXITIF (Dest <> 0)
								ENDLOOP ;/myLine loop
								EXITIF (Dest <> 0)
							ENDLOOP ;/myDepgh
						ENDIF ;/Dest = 0

						;Search for line with the most space
						;-----------------------------------
						IF (Dest = 0) THEN
							mySpace = 0
							myFound	= 0
							LOOP myLine = AreaStartLine TO AreaEndLine DO
								myLineValid = ((myLine >= MinLine) AND (myLine <= MaxLine))
								myLineUsed	= (D[myStartStop + myLine] > 0) ;Start / Stop On
								IF myLineValid AND myLineUsed THEN
									n 			= myLine
									SearchBag 	= (Line[n].LastBag)
									IF ((Bag[SearchBag].Prg = 0) AND (Line[n].Space > mySpace) AND Line[n].Clear) THEN
										;Found line with a matching program
										myFound	= n
										mySpace = Line[n].Space
									ENDIF ;/SearchBag
								ENDIF ;/myLineValid
							ENDLOOP ;/myLine loop

							IF (myFound > 0) THEN
								Dest 	= myFound
							ENDIF

						ENDIF ;/Dest = 0

					ENDIF ;/Area Valid
					EXITIF (Dest <> 0)
				ENDLOOP ;/Area Loop

			ENDIF ;/BufferDst > 0

			;Destination line found!!
			IF (Dest <> 0) THEN
				Buff = Buffer
				IF (Bag[myTransitBag].Cat = 0) AND (Bag[BufferBagNum[Buff]].Cat > 0) THEN ;Bag in Transit
					Bag[BufferBagNum[Buff]].Dst = USINT(Dest)
					Bag[myTransitBag]	= Bag[BufferBagNum[Buff]]
					Bag[BufferBagNum[Buff]]	 	= Bag[0]
					C[Dest] = 0
					D[900 + mySeq] 	= 3 ; Open buffer
				ENDIF
			ELSE
				;Storage full!!
				;Do Nothing? Alarm?
				;Other Area?
			ENDIF

		ENDIF ;/BagSettled

		;Buffer Alarms
		IF (BufferPrg > 0) AND NOT BufferSettled THEN
			Alarm[mySeq].Name 	= almBagNotAtProx
			Alarm[mySeq].Bag	= BufferBag
		ELSE IF (BufferPrg = 0) AND BufferSettled THEN
			Alarm[mySeq].Name 	= almBagNotShownOnScreen
			Alarm[mySeq].Bag	= BufferBag
		ENDIF
	ENDIF
ENDIF

;Clear Line Selections
LOOP n = 1 TO 5 DO
	LineSelect[n] = FALSE
ENDLOOP

;Step 3 - Select line / open buffer stop
IF (STEP = 3) THEN
	LineSelect[Dest] 	= TRUE
	Enable.SVC3LowLevel 		= (Buff = 1)
	Enable.SVC2FullBagLowLevel 	= (Buff = 2)
	;Bag arrived on selected line
	IF PLS THEN
		C[Dest] = 0
		IF (Bag[297].Cat = 0) AND (Bag[BufferBagNum[Buff]].Cat > 0) THEN
			Bag[297]				 	= Bag[BufferBagNum[Buff]]
			Bag[BufferBagNum[Buff]]	 	= Bag[0]
		ENDIF
	ENDIF

	;Bag released from SVC2
	IF ((Buff = 1) AND NOT Request.SVC2FullBagLowLevel) THEN
		D[912] = 4
	ENDIF

	;Bag released from SVC3
	IF ((Buff = 2) AND NOT Request.SVC3LowLevel) THEN
		D[912] = 4
	ENDIF
	Alarm[mySeq].Name = almBagNotArrived
ENDIF

;Step 4 - Select line / open buffer stop
IF (STEP = 4) THEN

	LineSelect[Dest] 			= TRUE

	;Bag arrived on selected line
	IF Line[Dest].Trip THEN
		D32[498] 				 	= Bag[297].Cus	;Set Customer for Customer FIFO
		Bag[297].Dst 				= 0 		    ;Clear Destination
		Bag[Line[Dest].LastBag] 	= Bag[297]
		Bag[297] 					= Bag[0]
		D[912] 						= 1
	ENDIF

	Alarm[12].Name = almBagNotArrived

ENDIF
;Alarms
TimerAlarm.IN = NOT PLS AND (Alarm[mySeq].Name > 0) AND (AlarmOld = Alarm[mySeq].Name)
TimerAlarm.PT = Alarm[mySeq].Time
TimerAlarm FUB TON_10ms()
Alarm[mySeq].On = TimerAlarm.Q
Alarm[mySeq].ET = TimerAlarm.ET

AlarmOld = Alarm[mySeq].Name ;Need to ensure alarm changes as may be multiple alarms on step 2

Enable.PN[1] = O_OpenBuffer[1]

;Outputs
Y[4].Y01 = LineSelect[1]
Y[4].Y02 = LineSelect[2]
Y[4].Y03 = LineSelect[3]
Y[4].Y04 = LineSelect[4]
Y[4].Y16 =  (O_Reset OR LineSelect[5])

END_PROGRAM
```

### Program Logical/Sequences/10ms/13_spf2 (IEC) - * Soiled Offgoing Transfer Lines 1 - 14

#### 5_spf1.var
```iecst
VAR RETAIN
	STEP : UINT;
	LASTSTEP : UINT;
	PLS : BOOL;
	BagSettledTime : ARRAY[0..99] OF UINT;
	Destination : UINT;
	SettleTime : UINT;
	BestTime : UINT;
	LineSelect : ARRAY[0..49] OF BOOL;
	ResetPointsET : TIME;
	ResetPoints : BOOL;
	n : UINT;
	IncSettle : BOOL;
	LineSettle : ARRAY[0..99] OF BOOL;
	I_BagAtStop : ARRAY[0..49] OF BOOL;
	OffGoingEnable : BOOL;
	AlarmBagNotProx : BOOL;
	SearchDest : UINT;
END_VAR
VAR
	TimerAlarm : TON_10ms;
	MaxBuffers : UINT;
	ResetBrush : BOOL;
	FoundLine : UINT;
	O_Reset : BOOL;
	O_SDCBufferOpen : ARRAY[0..4] OF BOOL;
	I_SDCBagAtBuffer : ARRAY[0..4] OF BOOL;
	ResetBrushET : TIME;
	SVC2BufferClear : BOOL;
	CloseBrush : BOOL;
	SDC4_Valid : BOOL;
	I_BagPassedSVC2 : BOOL;
	EnableSDC3Search : BOOL;
	EnableSDC1Search : BOOL;
	Alternator : UINT;
	LastDest : UINT;
	I_ApproachBrush : BOOL;
	O_CloseBrush : BOOL;
	SDC1_Valid : BOOL;
	SDC2_Valid : BOOL;
	SDC3_Valid : BOOL;
	EmptyInTransit : BOOL;
	CloseStop : BOOL;
	I_BagReleased : BOOL;
	BufferBag : ARRAY[0..4] OF UINT;
	BufferClear : ARRAY[0..4] OF BOOL;
	testAtStop : BOOL;
	PairingLoop : BOOL;
	LowLevelBufferClear : BOOL;
END_VAR
```

#### 5_spf1Cyclic.ab
```automation-basic
PROGRAM _CYCLIC
	(* cyclic program *)

;----------------------------------------
;Sequence 5 - SPF1 Offgoing Points D[905]
;----------------------------------------
;Inputs
;------

OffGoingEnable 		= ((D[26] > 0) AND NOT Std.HaltSys)

I_BagAtStop[1] 		= X[5].X01
I_BagAtStop[2] 		= X[5].X02
I_BagAtStop[3] 		= X[5].X03
I_BagAtStop[4] 		= X[5].X04
I_BagAtStop[5] 		= X[5].X05

O_Reset 			= FALSE

;Buffer line configuration
;-------------------------
MaxBuffers			= 2

BufferBag[1]		= 261 ;Last buffer bag number
BufferBag[2]		= 272 ;Last buffer bag number

BufferClear[1] 		= ((D[21] > 0)) ;AND (Bag[BufferBag[1]].Cat = 0) AND NOT O_SDCBufferOpen[1] AND NOT I_SDCBagAtBuffer[1])
BufferClear[2]		= ((D[22] > 0)) ;AND (Bag[BufferBag[2]].Cat = 0) AND NOT O_SDCBufferOpen[2] AND NOT I_SDCBagAtBuffer[2])

LowLevelBufferClear  = (NOT X[11].X06  AND NOT Y[11].Y06);LOW LEVEL SINGLE BAG BUFFER

;Alternating between SDC1 and SDC3

Uld[1].SDCReady 	= (BufferClear[1] ) ;Passed to unloading search
Uld[2].SDCReady 	= (BufferClear[2] );Passed to unloading search

Alarm[13].Name 		= 0
Alarm[13].Bag		= 324
Alarm[13].Beacon		= TRUE
Alarm[13].Extra		= 0
Alarm[13].Time		= 3000

;Setup Sequence
;--------------
STEP = D[913]
;Setup Pulse contact
PLS = (STEP <> LASTSTEP)
LASTSTEP = STEP

;Sequence Steps
;--------------
IF (STEP = 0) THEN
	;Disabled
ENDIF

;Step 1 - Reset Points
TON_10ms((STEP = 1),300,ResetPoints,ResetPointsET)
IF (STEP = 1) THEN
	O_Reset 	= TRUE
	FoundLine 	= 0
	Destination = 0
	;IF (ResetPoints AND OffGoingEnable) THEN
	IF (ResetPoints AND OffGoingEnable AND NOT I_BagReleased) THEN
		D[913] = 2
	ENDIF
ENDIF

;Bags on storage line timers
R_TRIG(Std.Clock100ms,IncSettle)
AlarmBagNotProx 	= FALSE
AlarmBagNotProxLine = 0

LOOP n = 1 TO 5 DO

	LineSettle[n]  = (I_BagAtStop[n] AND (Bag[Line[n].FirstBag].Cat > 0))
	IF IncSettle AND LineSettle[n] AND (BagSettledTime[n] < $FFFF) THEN
		BagSettledTime[n] = BagSettledTime[n] + 1
	ELSE IF NOT LineSettle[n] THEN
		BagSettledTime[n] = 0
		;If Bag has destiantion and not at stop then alarm
		IF (STEP = 2) AND (Bag[Line[n].FirstBag].Dst > 0) THEN
			Alarm[13].Name	= almBagNotAtProx
			Alarm[13].Bag	= Line[n].FirstBag
			Alarm[13].Extra 	= n
		ENDIF
	ENDIF

ENDLOOP

;Buffer trip not correct alarms
;LOOP n = 1 TO MaxBuffers DO
;	IF (STEP = 2) AND BufferClear[n] AND NOT Uld[n].SDCReady THEN
;		Alarm[5].Name 	= almSwitchFault
;		Alarm[5].Bag	= BufferBag[n]
;	ENDIF
;ENDLOOP

;Search for the bag with a valid destination that has been waiting the longest
IF STEP = 2 THEN

	FoundLine 	= 0
	Destination = 0
	BestTime 	= 0
	SettleTime = 30 ;3 seconds

	LOOP n = 1 TO 5 DO

		IF (BagSettledTime[n] > SettleTime) THEN
			SearchDest = Bag[Line[n].FirstBag].Dst

			SDC1_Valid  = ((SearchDest = 21) AND BufferClear[1])
			SDC2_Valid 	= ((SearchDest = 22) AND BufferClear[2])

			IF (SDC1_Valid OR SDC2_Valid ) THEN
				FoundLine 	= n
				Destination = SearchDest
				BestTime 	= BagSettledTime[n]
			ENDIF
		ENDIF

	ENDLOOP

	IF ((FoundLine > 0) AND OffGoingEnable AND (Bag[324].Cat = 0) AND Line[23].Clear AND (Bag[325].Cat = 0) AND LowLevelBufferClear) THEN
		C[23]  = 0
		D[913] = 3
	ENDIF

ENDIF

;Step 3 - Select Line / Open Stop, Until Bag at correct destination
;Clear Line Selections
LOOP n = 1 TO 5 DO
	LineSelect[n] = FALSE
	Indication[n] = FALSE
ENDLOOP

IF (STEP = 3) THEN

	IF PLS THEN
		C[23] = 0
	ENDIF

	IF (Bag[324].Cat = 0) AND (Bag[Line[FoundLine].FirstBag].Cat > 0)THEN
		Bag[324] 						= Bag[Line[FoundLine].FirstBag]
		Bag[Line[FoundLine].FirstBag] 	= Bag[0]
	ENDIF

	;Select Line - Wait for bag to arrive
	LineSelect[FoundLine] = TRUE ;TRUE
	Indication[FoundLine] = TRUE ;Use indication as single stop and display dosen't indicate to operator where the bag is comming from

	;Select Route
	IF (Destination = 21) OR (Destination = 22) THEN
		Uld[1].DischargerStartLine = FoundLine ;Unloading Program

		IF ((C[23] > 0) AND NOT PLS) THEN
			Uld[1].DischargerStartLine = FoundLine ;Unloading Program

			Bag[Line[23].LastBag] 	= Bag[324]
			Bag[324] 				= Bag[0]
			D[913] 					= 1
			ENDIF
		ENDIF

	Alarm[13].Name	= almBagNotReleased

ENDIF

;SSR2 Brush speed reducer

;Alarms
TimerAlarm.IN = NOT PLS AND (Alarm[13].Name > 0)
TimerAlarm.PT = Alarm[13].Time
TimerAlarm FUB TON_10ms()
Alarm[13].On = TimerAlarm.Q
Alarm[13].ET = TimerAlarm.ET

;Outputs
;-------
Y[5].Y16 = O_Reset

Y[5].Y01 = LineSelect[1]
Y[5].Y02 = LineSelect[2]
Y[5].Y03 = LineSelect[3]
Y[5].Y04 = LineSelect[4]
Y[5].Y05 = LineSelect[5]

END_PROGRAM
```

### Program Logical/Sequences/10ms/14_svc4 (IEC, version 1.00.0) - * SVC3 Vertical Conveyor

#### 18_svc3Cyclic.ab
```automation-basic
PROGRAM _CYCLIC
	(* cyclic program *)

;---------------------------------------------------
;Sequence 13 - SIC2 Soiled Incline Conveyor 2 D[913]
;---------------------------------------------------

;Inputs
I_CarrAtTop				= X[11].X01
I_CarrAtBottom			= X[11].X02
I_CarrAtFullBagInHigh   = X[11].X03
I_BagOnCarr				= X[11].X04

I_BagAtBufferStopHigh   = X[11].X05
I_BagAtBufferStopLow    = X[11].X06

O_OpenHighLevelBuffer	= FALSE
O_OpenLowLevelBuffer	= FALSE ;X[12].X15
O_OpenLowLevelBufferStop = FALSE

;I_BagAtLLBuff			= FALSE ;X[12].X01
;O_LLBuffOpen			= FALSE ;Y[12].Y01

O_OpenBuffer			= FALSE
O_MoveCarrUp			= FALSE
O_MoveCarrDown			= FALSE
OpenCarriageStop		= FALSE

Request.SVC4ToSDP1		= FALSE

Alarm[14].Name 			= 0
Alarm[14].Bag			= 319
Alarm[14].Beacon		= TRUE
Alarm[14].Extra			= 0
Alarm[14].Time			= 3000

;Setup Sequence
STEP = D[914]
;Setup Pulse contact
PLS = (STEP <> LASTSTEP)
LASTSTEP = STEP

;Sequence
IF (STEP = 0) THEN
	;Disabled
ENDIF

;Move carriage down from top position
IF (STEP = 1) THEN
	O_MoveCarrDown = NOT I_CarrAtFullBagInHigh
	IF I_CarrAtFullBagInHigh THEN
		D[914] = 2
	ENDIF
	IF NOT Std.EStop THEN
		Alarm[14].Name = almCarriageMoveFault
	ENDIF
ENDIF

;Check Status
IF (STEP = 2) THEN
	IF NOT I_BagOnCarr  THEN
		D[914] = 3
	ENDIF
	IF I_BagOnCarr THEN
		Alarm[14].Name = almSwitchFault
	ENDIF
ENDIF

;Wait for bag at buffer or bag in transit to High or Low buffer
TON_10ms((I_BagAtBufferStopHigh AND (Bag[320].Cat > 0)),300,SettledHighLevelBuffer,SettledHighLevelBufferET)
TON_10ms((I_BagAtBufferStopLow AND (Bag[325].Cat > 0)),300,SettledLowLevelBuffer,SettledLowLevelBufferET)
IF (STEP = 3) THEN

	IF SettledHighLevelBuffer  THEN
		D[914] = 4
	ELSE IF SettledLowLevelBuffer OR (Bag[324].Cat > 0) THEN
		D[914] = 10 ;move carriage down to SDP1
	ENDIF

ENDIF

;Open Buffer stop - Enable
IF (STEP = 4) THEN
	O_OpenHighLevelBuffer 	= (NOT I_BagOnCarr AND I_CarrAtFullBagInHigh)
	;Enable.SVC[2] 	= (NOT I_BagOnCarr AND I_CarrAtTop)
	IF ((Bag[319].Cat = 0) AND (Bag[320].Cat > 0)) THEN
		Bag[319] = Bag[320]
		Bag[320] = Bag[0]
	ENDIF
	IF I_BagOnCarr THEN
		D[914] = 5
	ENDIF
	Alarm[14].Name = almBagNotArrived
ENDIF

;Let bag settle on carriage
TON_10ms(I_BagOnCarr,300,BagSettledOnCarr,BagSettledOnCarrET)
IF (STEP = 5) THEN
	IF ((Bag[319].Dst = 21) AND BagSettledOnCarr AND NOT I_CarrAtTop) THEN
		D[914] = 6
	ELSE IF ((Bag[319].Dst = 22) AND BagSettledOnCarr AND NOT I_CarrAtBottom) THEN
		D[914] = 10
	ENDIF
	Alarm[14].Name = almBagNotSettled
ENDIF

;Move Carriage up to carriage at top
IF (STEP = 6) THEN
	O_MoveCarrUp = NOT I_CarrAtTop
	IF I_CarrAtTop THEN
		D[914] = 7
	ENDIF
ENDIF

;check buffer clear
IF (STEP = 7) THEN

	IF (Line[21].Clear AND (Bag[356].Cat = 0) AND(Bag[269].Cat = 0)) THEN
		C[21]  = 0
		C[31]  = 0
		D[914] = 8
	ENDIF
	IF NOT Std.EStop THEN
		Alarm[14].Name = almCarriageMoveFault
	ENDIF
ENDIF

;open carriage stop
IF (STEP = 8) THEN
	IF PLS THEN
		C[31] = 0
	ENDIF

	;IF (Line[33].Clear AND NOT I_BagAtLLBuff AND NOT O_LLBuffOpen AND NOT Std.HaltSys) THEN
	OpenCarriageStop = I_CarrAtTop
	IF ((Bag[269].Cat = 0) AND (Bag[319].Cat > 0)) THEN
		Bag[319].Dst = 0
		Bag[269]     = Bag[319]
		Bag[319]     = Bag[0]
	ENDIF

	IF Line[31].Clear THEN
		D[914] = 9
	ENDIF
	;IF NOT Std.HaltSysLoading THEN
		;IF X[11].X07 OR  THEN
	;		Alarm[14].Name = almBagNotReleased
		;ENDIF
;	ENDIF
ENDIF

;VC4 Bag in transit
IF (Bag[269].Cat > 0) THEN
	IF (Line[21].Trip AND (Bag[356].Cat = 0)) THEN
		Bag[356] = Bag[269]
		Bag[269] = Bag[0]
	ENDIF
	Alarm[14].Bag	= 269
	Alarm[14].Name 	= almBagNotArrived
ENDIF

;check status
IF (STEP = 9) THEN
	IF NOT I_CarrAtFullBagInHigh AND NOT I_BagOnCarr THEN
		D[914] = 1
	ENDIF

	IF NOT Std.EStop THEN
		Alarm[14].Name = almSwitchFault
	ENDIF
ENDIF

;move down to low level
IF (STEP = 10) THEN
	O_MoveCarrDown = NOT I_CarrAtBottom
	IF (I_CarrAtBottom AND (Bag[319].Cat > 0))THEN
		D[914] = 11
		ELSE IF (I_CarrAtBottom AND (Bag[319].Cat = 0))THEN
		D[914] = 13
	ENDIF
	Alarm[14].Name = almCarriageMoveFault
ENDIF

;carriage at bottom
;IF (STEP = 11) THEN
;	IF I_CarrAtBottom THEN
;		D[914] = 12
;	ENDIF
;ENDIF

;Check SDP1
IF (STEP = 11) THEN
	Request.SVC4ToSDP1 = I_CarrAtBottom
	IF Enable.SVC4ToSDP1 THEN

		D[914] = 12
	ENDIF
ENDIF

;Open carriage stop
IF (STEP = 12) THEN
	OpenCarriageStop  = I_CarrAtBottom
	IF ((Bag[319].Cat > 0) AND (Bag[285].Cat > 0)) THEN
		Bag[285] = Bag[319]
		Bag[319] = Bag[0]
	ENDIF
	IF NOT Enable.SVC4ToSDP1 THEN
		D[914] = 13
	ENDIF
ENDIF

;check buffers
IF (STEP = 13) THEN
	IF SettledHighLevelBuffer  THEN
		D[914] = 16
	ELSE IF SettledLowLevelBuffer OR (Bag[324].Cat > 0) THEN
		D[914] = 14 ;
	ENDIF
ENDIF

;open low level buffer stop
IF (STEP = 14) THEN
	O_OpenLowLevelBufferStop = I_CarrAtBottom

	IF ((Bag[325].Cat > 0) AND (Bag[319].Cat = 0)) THEN
		Bag[319] = Bag[325]
		Bag[325] = Bag[0]
	ENDIF

	IF I_BagOnCarr THEN
		D[914] = 15
	ENDIF
	Alarm[14].Name = almBagNotArrived
ENDIF

;decide where bag is going
IF (STEP = 15) THEN
	IF BagSettledOnCarr THEN
		IF Bag[319].Dst = 22 THEN
			D[914] = 11
		ELSE IF Bag[319].Dst = 21 THEN
			D[914] = 6
		ENDIF
	ENDIF
ENDIF

;move up
IF (STEP = 16) THEN
	O_MoveCarrUp = NOT I_CarrAtTop
	IF I_CarrAtFullBagInHigh THEN
		D[914] = 17
	ENDIF
ENDIF

;move carriage passed full bag in height
TON_10ms(NOT I_CarrAtFullBagInHigh,50,CarriagePassed,CarriagePassedET)
IF (STEP = 17) THEN
	O_MoveCarrUp = NOT I_CarrAtTop
	IF CarriagePassed THEN

		D[914] = 1
	ENDIF
ENDIF

;Alarms
TimerAlarm.IN 	= NOT PLS AND (Alarm[14].Name > 0)
TimerAlarm.PT 	= Alarm[13].Time
TimerAlarm FUB TON_10ms()
Alarm[14].On 	= TimerAlarm.Q
Alarm[14].ET 	= TimerAlarm.ET

;Inverter Speed Selections
;-------------------------
;High Speed Used For Up		= 50Hz
;Medium Speed Used For Down	= 50Hz

;TON_10ms(O_MoveCarrUp,500,HighSpeedUp,HighSpeedUpET)
;TON_10ms(O_MoveCarrDown,500,HighSpeedDn,HighSpeedDnET)
;IF (STEP = 4) THEN
;	Y[3].Y14 = (NOT HighSpeedUp) 							;High Speed
;	Y[3].Y15 = FALSE										;Medium Speed
;ELSE IF (STEP = 7) THEN
;;	Y[3].Y14 = FALSE										;High Speed
;	Y[3].Y15 = (NOT HighSpeedDn)							;Medium Speed
;ELSE
;	Y[3].Y14 = FALSE
;	Y[3].Y15 = FALSE
;ENDIF

;PLC Outputs
;-----------
Y[11].Y05 		= O_OpenHighLevelBuffer
Y[11].Y06       = O_OpenLowLevelBufferStop
Y[13].Y13 		= (O_MoveCarrUp 	AND NOT I_CarrAtTop) ;WASY1213
;Y[12].Y14 		= (O_MoveCarrDown AND NOT I_CarrAtBottom)
Y[13].Y15 		= O_MoveCarrDown ;WAS Y1215

;ReleaseBrake 	= (Y[8].Y06 OR Y[8].Y07)
;Y[8].Y09 		= ReleaseBrake
Y[13].Y16 		= OpenCarriageStop ;WAS Y1216

;Don't allow forcing of carriage movement and carriage stop
YForceDisable[12].Y13 = TRUE
;YForceDisable[12].Y14 = TRUE
YForceDisable[12].Y16 = TRUE
YForceDisable[12].Y15 = TRUE

;Don't allow forcing of carriage movement and carriage stop
YForceDisable[12].Y09 = TRUE
YForceDisable[12].Y06 = TRUE
YForceDisable[12].Y07 = TRUE
YForceDisable[12].Y12 = TRUE

END_PROGRAM
```

#### 18_svc3.var
```iecst
VAR RETAIN
	STEP : UINT;
	PLS : BOOL;
	LASTSTEP : UINT;
	O_OpenBufferStop : BOOL;
	I_BagAtBuffer : BOOL;
	O_RunMotor : BOOL;
	BagSettled : BOOL;
	BagSettledET : TIME;
	BagAtBuffer : BOOL;
	RunOnET : TIME;
	RunOn : BOOL;
	BagNearTopET : TIME;
	BagNearTop : BOOL;
	BagAtBufferET : UDINT;
	I_BagInIncline : BOOL;
END_VAR
VAR
	I_BagAtOutgoingBuffer : BOOL;
	zzTON_10ms00002 : TON_10ms;
	zzTON_10ms00003 : TON_10ms;
	I_PaddleInPosition : BOOL;
	zzTON_10ms00004 : TON_10ms;
	CloseBufferStop : BOOL;
	CloseBufferStopET : TIME;
	O_OutgoingBufferOpen : BOOL;
	TimerAlarm : TON_10ms;
	O_SelectSP4ToSP2 : BOOL;
	I_BagReleased : BOOL;
	O_SelectSP4 : BOOL;
	I_BagOutAtTop : BOOL;
	I_BagOutAtBottom : BOOL;
	I_BagOnCarriage : BOOL;
	I_CarriageAtTop : BOOL;
	I_CarriageAtBottom : BOOL;
	O_OpenCarriageStop : BOOL;
	O_MoveUp : BOOL;
	O_MoveDown : BOOL;
	I_BagAtBufferStop : BOOL;
	BagSettledAtBuffer : BOOL;
	BagSettledAtBufferET : TIME;
	BufferClear : BOOL;
	I_BagOutAtTopSVC3 : BOOL;
	I_CarrAtTop : BOOL;
	I_CarrAtBottom : BOOL;
	I_CarrAtFullBagIn : BOOL;
	I_BagOnCarr : BOOL;
	O_SP1Bend : BOOL;
	O_SP3Straight : BOOL;
	O_SP8Bend : BOOL;
	O_OpenBuffer : BOOL;
	O_MoveCarrUp : BOOL;
	O_MoveCarrDown : BOOL;
	O_OpenCarrStop : BOOL;
	O_SP3Bend : BOOL;
	SettledBuffer : BOOL;
	SettledBufferET : UDINT;
	ParingLoopEnabled : BOOL;
	BagSettledOnCarr : BOOL;
	BagSettledOnCarrET : UDINT;
	PairOnLoop : BOOL;
	PairNotValidSVC3 : BOOL;
	HLBagMatch : BOOL;
	NoPairForSVC3 : BOOL;
	LLBagMatch : BOOL;
	CarriagePasted : BOOL;
	CarriagePastedET : UDINT;
	I_CarrAtFullBagInHigh : BOOL;
	I_BagAtBufferStopHigh : BOOL;
	I_BagAtBufferStopLow : BOOL;
	OpenCarriageStop : BOOL;
	SettledHighLevelBuffer : BOOL;
	SettledHighLevelBufferET : UDINT;
	SettledLowLevelBuffer : BOOL;
	SettledLowLevelBufferET : UDINT;
	O_OpenHighLevelBuffer : BOOL;
	O_OpenLowLevelBuffer : BOOL;
	O_OpenLowLevelBufferStop : BOOL;
	CarriagePassed : BOOL;
	CarriagePassedET : UDINT;
END_VAR
```

### Program Logical/Sequences/10ms/15_sdp (IEC) - * SDC1 Machine 1 BIN/BCD

#### 6_sdc1.var
```iecst
VAR RETAIN
	STEP : UINT;
	PLS : BOOL;
	LASTSTEP : UINT;
	SteadyUp : BOOL;
	CloserUpET : TIME;
	SteadysDown : BOOL;
	SteadysDownET : TIME;
	LoadDropped : BOOL;
	SteadyUpET : TIME;
	CloserDownET : TIME;
	SettledAtDischargerET : TIME;
	MinOpenET : TIME;
	SettledAtDischarger : BOOL;
	CloserDown : BOOL;
	MinOpen : BOOL;
	CloserUp : BOOL;
	SettledAtBuffer : BOOL;
	SettledAtBufferET : TIME;
	I_BagAtBuffer : BOOL;
	O_OpenStop : BOOL;
	O_OpenBag : BOOL;
	O_Steadys : BOOL;
	O_OpenBuffer : BOOL;
	O_Closer : BOOL;
	I_BagAtDischarger : BOOL;
	I_OpenBag : BOOL;
	I_LoadDropped : BOOL;
	TestDrop : BOOL;
END_VAR
VAR
	DischargerEnable : BOOL;
	TestDischarger : BOOL;
	I_BagEmpty : BOOL;
	O_BagReady : BOOL;
	I_BagReleased : BOOL;
	O_EmptyBagBufferOpen : BOOL;
	I_BagAtEmptyBuffer : BOOL;
	TimerAlarm : TON_10ms;
	CodeStep : BOOL;
	BCD_BIN_CAT : BCD_BIN_OUTPUT;
	BCD_BIN_CUS : BCD_BIN_OUTPUT;
	BCD_BIN_WGT : BCD_BIN_OUTPUT;
	Remainder : UINT;
	WgtRound : UINT;
	HaltDownStairs : BOOL;
	O_StaticBag : BOOL;
	OpenStatic : BOOL;
	OpenStaticET : UDINT;
END_VAR
```

#### 6_sdc1Cyclic.ab
```automation-basic
PROGRAM _CYCLIC
	(* cyclic program *)

;Sequence 6 - Discharger 1 D[906]

;-----------------------------------------
;Revision 1.00 19/12/2005 D.J. First Issue
;-----------------------------------------

DischargerEnable 		= ((D[23] > 0) AND NOT Std.HaltSys)

I_BagAtDischarger		= X[8].X01
I_OpenBag				= CAN[1].DropLoad
I_LoadDropped			= X[8].X16
I_BagReleased			= FALSE ;X[6].X02
I_BagEmpty			  	= TRUE
HaltDownStairs          = NOT X[6].X12

O_BagReady				= FALSE
O_StaticBag 			= FALSE
O_Steadys				= FALSE
O_Closer				= FALSE
O_OpenBag				= FALSE
O_OpenStop				= FALSE

Enable.SVC4ToSDP1 		= FALSE
Request.SDP[1]          = FALSE

;Alarm
Alarm[15].Name 			= almNoAlarm ;Clear sequence alarm name
Alarm[15].Bag 			= 285
Alarm[15].Beacon		= TRUE
Alarm[15].Extra			= 0
Alarm[15].Time			= 3000

;Setup Sequence
STEP = D[915]
;Setup Pulse contact
PLS = (STEP <> LASTSTEP)
LASTSTEP = STEP

;Step 0 - Disabled
IF (STEP = 0) THEN
	;Disabled
ENDIF

;Check Status - No bag at discharger,  and no bag at discharger on the screen
;TON_10ms(I_BagAtBuffer,300,SettledAtBuffer,SettledAtBufferET)
IF (STEP = 1) THEN
	IF (DischargerEnable  AND NOT I_BagAtDischarger AND (Bag[285].Cat = 0)  AND NOT HaltDownStairs) THEN
		IF Request.SVC4ToSDP1 THEN
			D[915] = 2
		ENDIF
	ENDIF
	IF (Bag[285].Cat > 0) THEN
		Alarm[15].Name = almBagDataError
	ELSE IF I_BagAtDischarger THEN
		Alarm[15].Name = almSwitchFault
	;ELSE IF (Bag[285].Cat > 0) AND NOT I_BagAtBuffer THEN
	;	Alarm[6].Name 	= almBagNotAtProx
	;	Alarm[6].Bag	= 285
	;ELSE IF (Bag[285].Cat = 0) AND I_BagAtBuffer THEN
	;	Alarm[6].Name 	= almBagNotShownOnScreen
	;	Alarm[6].Bag	= 285
	ENDIF
ENDIF

;Wait for bag in discharger
IF (STEP = 2) THEN
	Enable.SVC4ToSDP1 	= TRUE
	;Enable.SDC[1] 	= TRUE
	IF I_BagAtDischarger THEN
		D[915] = 3
	ENDIF
	Alarm[15].Name = almBagNotArrived
ENDIF

;Let bag settle in discharger
TON_10ms(((STEP = 3)AND I_BagAtDischarger),600,SettledAtDischarger,SettledAtDischargerET)
IF (STEP = 3) THEN

	IF (Bag[285].Cat = 0) AND (Bag[319].Cat > 0) THEN
		Bag[285] = Bag[319]
		Bag[319] = Bag[0]
	ENDIF
	IF SettledAtDischarger THEN
		D[915] = 4
	ENDIF
	Alarm[15].Name = almBagNotSettled
ENDIF

;Allow steadys to move down
TON_10ms((STEP = 4),400,SteadysDown,SteadysDownET)
IF (STEP = 4) THEN
	IF SteadysDown THEN
		D[915] = 5
	ENDIF
	IF (Bag[285].Cat = Std.MaxCats) THEN
		D[915] = 8
	ENDIF
ENDIF

;Steady cylinders on from steps 4 - 9
O_Steadys = ((STEP >= 4) AND (STEP <= 9))

;Bag opener on from step 5 - 8
O_OpenBag = ((STEP >= 6) AND (STEP <= 8))

CodeStep  = ((STEP >= 4) AND (STEP <= 5))

;Bag Ready to Washing Machine
IF (STEP = 5) THEN
	;Request.SDP[1] = TRUE
	;CAN[1].BagReady = TRUE
	IF NOT Y[8].Y05 AND NOT HaltDownStairs THEN
		D[915] = 6
	ENDIF

ENDIF

;Set LoadDropped to False
IF (STEP <> 6) THEN
	LoadDropped = FALSE
ENDIF

;Open Bag Until LoadDropped recieved and has been open for 6 seconds
TON_10ms((STEP = 6),600,MinOpen,MinOpenET) ;ET means Elapsed Time
IF (STEP = 6) THEN

	Request.SDP[1] = MinOpen
	O_OpenBag      = TRUE

	;IF (LoadDropped AND MinOpen) THEN
		;Write Report
		;------------
		;IF (ReportUnloading[1].Cat = 0) THEN
		;	ReportUnloading[1].Cat = UINT(Bag[260].Cat)	;Category
		;	ReportUnloading[1].Cus = Bag[260].Cus		;Customer
		;	ReportUnloading[1].Wgt = Bag[260].Wgt		;Weight
		;	ReportUnloading[1].Cnt = 0					;Count
		;	ReportUnloading[1].Stn = 0					;Station
		;	ReportUnloading[1].Mcn = 1					;Machine
		;ENDIF
	;ENDIF
	IF  MinOpen AND Enable.SDP[1] AND NOT HaltDownStairs  THEN

		IF ((Bag[285].Cat > 0) AND (Bag[287].Cat > 0)) THEN
			Bag[287].Wgt = Bag[285].Wgt + Bag[287].Wgt
		ELSE IF ((Bag[285].Cat > 0) AND (Bag[287].Cat = 0)) THEN
			Bag[287] = Bag[285]
			Bag[285] = Bag[0]
		ENDIF

		D[915] = 7
	ENDIF
	Alarm[15].Name = almLoadNotDropped
ENDIF

;Change display to empty bag
TON_10ms((STEP = 7),600,OpenStatic,OpenStaticET) ;ET means Elapsed Time
IF (STEP = 7) THEN
	O_StaticBag = Request.LU[2]
	IF OpenStatic AND NOT Enable.SDP[1] AND NOT HaltDownStairs THEN
		Bag[285].Cat 	= Std.MaxCats
		;Bag[287]        = Bag[286]
		;Bag[287]        = Bag[0]
		D[915] 			= 8
	ENDIF
	Alarm[15].Name = almGeneralSequence
ENDIF

;Close bag
TON_10ms((STEP = 8),800,CloserDown,CloserDownET)
IF (STEP = 8) THEN
	O_Closer = TRUE
	IF CloserDown THEN
		D[915] = 9
	ENDIF
ENDIF

;Allow closer to go back up
TON_10ms((STEP = 9),300,CloserUp,CloserUpET)
IF (STEP = 9) THEN
	IF CloserUp THEN
		D[915] = 10
	ENDIF
ENDIF

;Allow steadys to go up
TON_10ms((STEP = 10),200,SteadyUp,SteadyUpET)
IF (STEP = 10) THEN
	IF SteadyUp  THEN
		D[915] = 11
	ENDIF
ENDIF

;Check for space on empty bag buffer / Request release
IF (STEP = 11) THEN

	IF Request.EmptyBagInSVC[5] AND NOT X[8].X02 THEN
		D[915] = 12
	ENDIF
ENDIF

;Open buffer stop - unitl bag out
IF (STEP = 12) THEN
	O_OpenStop = TRUE
	;IF PLS THEN
	;	C[24] = 0
	;ENDIF
	Bag[285].Cat = 0
	Bag[285].Cus = 0
	Bag[285].Wgt = 0
	IF X[8].X02 THEN
		D[915] = 1
	ENDIF
	Alarm[15].Name = almBagNotReleased
ENDIF

;Alarms
TimerAlarm.IN 	= NOT PLS AND (Alarm[15].Name > 0)
TimerAlarm.PT 	= Alarm[15].Time
TimerAlarm FUB TON_10ms()
Alarm[15].On 	= TimerAlarm.Q
Alarm[15].ET 	= TimerAlarm.ET

;Outputs
;Y[24].Y16 	= O_BagReady
;Y[6].Y01 	= O_OpenBuffer
Y[8].Y01 	= O_Steadys
Y[8].Y02 	= O_OpenBag
Y[8].Y04 	= O_Closer
Y[8].Y03 	= O_OpenStop
Y[8].Y05    = O_StaticBag
END_PROGRAM
```

### Program Logical/Sequences/10ms/18_sic_1 (IEC) - * SP2 Empty bags from SDC1/2

#### 12_sp2.var
```iecst
VAR RETAIN
	STEP : UINT;
	PLS : BOOL;
	LASTSTEP : UINT;
END_VAR
VAR
	TimerAlarm : TON_10ms;
	I_BagAtBuffer : BOOL;
	O_OpenBuffer : BOOL;
	SDC2BufferFullET : TIME;
	SDC2BufferFull : BOOL;
	SettledBufferET : TIME;
	SettledBuffer : BOOL;
	O_OpenSP2BufferStop : BOOL;
	O_SelectPoint : BOOL;
	SP2BufferFull : BOOL;
	SP2BufferFullET : UDINT;
	ParingLoopEnabled : BOOL;
	BagInLoopHasDest : BOOL;
	O_OpenSDC1BufferStop : BOOL;
	BagSettledAtBuffer : BOOL;
	BagSettledAtBufferET : UDINT;
	Alternator : USINT;
	I_PaddleInPosition : BOOL;
	I_BagInIncline : BOOL;
	O_OpenBufferStop : BOOL;
	O_RunMotor : BOOL;
	I_BagAtOutgoingBuffer : BOOL;
	O_OutgoingBufferOpen : BOOL;
	BagSettled : BOOL;
	BagSettledET : UDINT;
	BagNearTop : BOOL;
	BagNearTopET : UDINT;
	CloseBufferStop : BOOL;
	CloseBufferStopET : UDINT;
	RunOn : BOOL;
	RunOnET : UDINT;
END_VAR
```
